C03656=1197.588,180.160,-56.490,-177.893,6.359,148.532
C03657=1197.583,180.408,-56.512,-177.890,6.361,148.532
C03658=1197.578,180.657,-56.536,-177.888,6.363,148.532
C03659=1197.574,180.906,-56.558,-177.885,6.365,148.531
C03660=1197.569,181.155,-56.581,-177.882,6.367,148.531
C03661=1197.565,181.403,-56.603,-177.880,6.368,148.531
C03662=1197.560,181.653,-56.626,-177.877,6.370,148.530
C03663=1197.555,181.902,-56.649,-177.874,6.372,148.530
C03664=1197.551,182.151,-56.672,-177.871,6.373,148.529
C03665=1197.546,182.400,-56.694,-177.868,6.375,148.529
C03666=1197.542,182.648,-56.717,-177.866,6.377,148.529
C03667=1197.537,182.898,-56.740,-177.864,6.378,148.528
C03668=1197.533,183.146,-56.763,-177.861,6.380,148.528
C03669=1197.527,183.395,-56.786,-177.858,6.382,148.527
C03670=1197.523,183.644,-56.809,-177.856,6.383,148.527
C03671=1197.519,183.893,-56.832,-177.853,6.385,148.527
C03672=1197.514,184.142,-56.855,-177.850,6.387,148.526
C03673=1197.509,184.392,-56.878,-177.848,6.389,148.526
C03674=1197.504,184.661,-56.902,-177.845,6.391,148.526
C03675=1197.499,184.930,-56.928,-177.842,6.393,148.525
C03676=1197.495,185.200,-56.952,-177.839,6.395,148.525
C03677=1197.489,185.469,-56.977,-177.836,6.397,148.525
C03678=1197.484,185.718,-57.000,-177.834,6.399,148.524
C03679=1197.480,185.967,-57.022,-177.831,6.400,148.524
C03680=1197.475,186.216,-57.046,-177.828,6.402,148.524
C03681=1197.470,186.465,-57.069,-177.826,6.404,148.523
C03682=1197.466,186.714,-57.092,-177.823,6.406,148.523
C03683=1197.462,186.963,-57.115,-177.820,6.408,148.523
C03684=1197.457,187.211,-57.138,-177.818,6.409,148.522
C03685=1197.452,187.460,-57.162,-177.815,6.411,148.522
C03686=1197.448,187.709,-57.184,-177.812,6.413,148.522
C03687=1197.443,187.958,-57.208,-177.810,6.415,148.521
C03688=1197.438,188.207,-57.231,-177.807,6.417,148.521
C03689=1197.434,188.456,-57.254,-177.805,6.419,148.520
C03690=1197.429,188.705,-57.278,-177.802,6.420,148.520
C03691=1197.424,188.953,-57.300,-177.799,6.422,148.520
C03692=1197.420,189.202,-57.324,-177.797,6.423,148.519
C03693=1197.415,189.451,-57.347,-177.794,6.425,148.519
C03694=1197.410,189.700,-57.370,-177.792,6.427,148.519
C03695=1197.406,189.949,-57.394,-177.789,6.429,148.518
C03696=1197.402,190.198,-57.416,-177.786,6.430,148.518
C03697=1197.397,190.447,-57.440,-177.784,6.432,148.518
C03698=1197.392,190.696,-57.463,-177.781,6.434,148.517
C03699=1197.388,190.945,-57.486,-177.779,6.436,148.517
C03700=1197.382,191.193,-57.509,-177.776,6.438,148.517
C03701=1197.378,191.442,-57.533,-177.774,6.440,148.516
C03702=1197.374,191.691,-57.556,-177.771,6.442,148.516
C03703=1197.369,191.940,-57.579,-177.768,6.443,148.516
C03704=1197.365,192.189,-57.603,-177.766,6.445,148.515
C03705=1197.360,192.438,-57.626,-177.763,6.447,148.515
C03706=1197.355,192.687,-57.650,-177.760,6.449,148.515
C03707=1197.350,192.936,-57.673,-177.758,6.451,148.514
C03708=1197.346,193.185,-57.696,-177.755,6.452,148.514
C03709=1197.341,193.434,-57.720,-177.752,6.454,148.514
C03710=1197.337,193.682,-57.744,-177.750,6.456,148.513
C03711=1197.332,193.931,-57.767,-177.747,6.458,148.513
C03712=1197.328,194.180,-57.790,-177.744,6.460,148.513
C03713=1197.323,194.429,-57.813,-177.742,6.461,148.512
C03714=1197.319,194.678,-57.837,-177.739,6.464,148.512
C03715=1197.314,194.926,-57.861,-177.736,6.466,148.512
C03716=1197.310,195.175,-57.884,-177.734,6.468,148.511
C03717=1197.305,195.425,-57.907,-177.731,6.470,148.511
C03718=1197.300,195.673,-57.932,-177.728,6.472,148.511
C03719=1197.296,195.922,-57.955,-177.726,6.473,148.510
C03720=1197.291,196.171,-57.978,-177.723,6.475,148.510
C03721=1197.287,196.419,-58.002,-177.720,6.477,148.510
C03722=1197.282,196.668,-58.026,-177.718,6.479,148.509
C03723=1197.277,196.917,-58.049,-177.715,6.481,148.509
C03724=1197.273,197.166,-58.073,-177.712,6.483,148.509
C03725=1197.268,197.415,-58.096,-177.710,6.484,148.508
C03726=1197.263,197.664,-58.120,-177.708,6.486,148.508
C03727=1197.259,197.912,-58.144,-177.705,6.488,148.508
C03728=1197.254,198.161,-58.167,-177.702,6.490,148.507
C03729=1197.250,198.410,-58.191,-177.700,6.492,148.507
C03730=1197.245,198.659,-58.215,-177.697,6.494,148.507
C03731=1197.240,198.908,-58.239,-177.694,6.496,148.506
C03732=1197.235,199.157,-58.263,-177.692,6.497,148.506
C03733=1197.231,199.406,-58.286,-177.689,6.499,148.506
C03734=1197.226,199.654,-58.310,-177.686,6.501,148.505
C03735=1197.222,199.904,-58.334,-177.684,6.503,148.505
C03736=1197.218,200.152,-58.358,-177.682,6.505,148.505
C03737=1197.213,200.401,-58.381,-177.679,6.507,148.505
C03738=1197.209,200.650,-58.405,-177.676,6.509,148.504
C03739=1197.204,200.899,-58.429,-177.673,6.511,148.504
C03740=1197.199,201.147,-58.453,-177.670,6.513,148.504
C03741=1197.194,201.396,-58.477,-177.668,6.515,148.503
C03742=1197.190,201.645,-58.501,-177.665,6.517,148.503
C03743=1197.185,201.893,-58.525,-177.662,6.518,148.503
C03744=1197.181,202.142,-58.548,-177.660,6.521,148.502
C03745=1197.177,202.391,-58.573,-177.658,6.522,148.502
C03746=1197.171,202.641,-58.597,-177.655,6.524,148.502
C03747=1197.167,202.889,-58.621,-177.652,6.526,148.501
C03748=1197.163,203.138,-58.645,-177.650,6.528,148.501
C03749=1197.158,203.387,-58.668,-177.647,6.530,148.501
C03750=1197.154,203.635,-58.692,-177.644,6.531,148.500
C03751=1197.149,203.884,-58.717,-177.642,6.534,148.500
C03752=1197.144,204.133,-58.741,-177.639,6.535,148.500
C03753=1197.140,204.382,-58.765,-177.636,6.538,148.500
C03754=1197.136,204.630,-58.789,-177.634,6.540,148.499
C03755=1197.130,204.880,-58.813,-177.631,6.542,148.499
C03756=1197.126,205.128,-58.837,-177.628,6.544,148.499
C03757=1197.122,205.377,-58.861,-177.626,6.545,148.498
C03758=1197.117,205.626,-58.885,-177.623,6.548,148.498
C03759=1197.112,205.875,-58.909,-177.621,6.549,148.498
C03760=1197.108,206.123,-58.933,-177.618,6.551,148.497
C03761=1197.103,206.372,-58.957,-177.615,6.553,148.497
C03762=1197.099,206.621,-58.983,-177.613,6.555,148.497
C03763=1197.094,206.870,-59.006,-177.610,6.557,148.496
C03764=1197.090,207.119,-59.030,-177.607,6.559,148.496
C03765=1197.085,207.367,-59.055,-177.605,6.561,148.496
C03766=1197.080,207.616,-59.079,-177.602,6.563,148.496
C03767=1197.076,207.865,-59.103,-177.599,6.565,148.495
C03768=1197.071,208.114,-59.127,-177.597,6.567,148.495
C03769=1197.067,208.363,-59.151,-177.594,6.569,148.495
C03770=1197.062,208.611,-59.175,-177.592,6.570,148.494
C03771=1197.058,208.860,-59.200,-177.589,6.573,148.494
C03772=1197.053,209.109,-59.224,-177.587,6.574,148.494
C03773=1197.048,209.358,-59.249,-177.583,6.577,148.494
C03774=1197.044,209.606,-59.273,-177.581,6.579,148.493
C03775=1197.040,209.855,-59.298,-177.578,6.581,148.493
C03776=1197.035,210.104,-59.322,-177.576,6.583,148.493
C03777=1197.030,210.352,-59.346,-177.573,6.585,148.492
C03778=1197.025,210.623,-59.372,-177.571,6.587,148.492
C03779=1197.020,210.894,-59.399,-177.568,6.589,148.492
C03780=1197.015,211.164,-59.426,-177.565,6.591,148.491
C03781=1197.010,211.434,-59.453,-177.562,6.594,148.491
C03782=1197.006,211.683,-59.477,-177.559,6.595,148.491
C03783=1197.002,211.932,-59.501,-177.556,6.597,148.490
C03784=1196.997,212.181,-59.526,-177.554,6.599,148.490
C03785=1196.992,212.429,-59.550,-177.552,6.601,148.490
C03786=1196.988,212.678,-59.575,-177.549,6.603,148.490
C03787=1196.983,212.927,-59.599,-177.546,6.606,148.489
C03788=1196.978,213.175,-59.624,-177.543,6.608,148.489
C03789=1196.975,213.425,-59.648,-177.540,6.609,148.489
C03790=1196.969,213.673,-59.673,-177.538,6.612,148.489
C03791=1196.965,213.921,-59.698,-177.536,6.613,148.488
C03792=1196.961,214.171,-59.723,-177.533,6.615,148.488
C03793=1196.956,214.419,-59.747,-177.530,6.617,148.488
C03794=1196.951,214.668,-59.771,-177.528,6.620,148.487
C03795=1196.947,214.917,-59.797,-177.525,6.622,148.487
C03796=1196.942,215.166,-59.821,-177.522,6.624,148.487
C03797=1196.938,215.415,-59.846,-177.520,6.625,148.486
C03798=1196.934,215.663,-59.870,-177.517,6.627,148.486
C03799=1196.929,215.911,-59.895,-177.515,6.629,148.486
C03800=1196.924,216.161,-59.920,-177.512,6.632,148.486
C03801=1196.920,216.409,-59.944,-177.509,6.634,148.485
C03802=1196.915,216.658,-59.970,-177.506,6.636,148.485
C03803=1196.911,216.907,-59.994,-177.504,6.638,148.485
C03804=1196.906,217.155,-60.019,-177.501,6.640,148.485
C03805=1196.901,217.405,-60.044,-177.499,6.642,148.484
C03806=1196.897,217.652,-60.069,-177.496,6.644,148.484
C03807=1196.893,217.902,-60.094,-177.493,6.646,148.484
C03808=1196.888,218.151,-60.118,-177.491,6.648,148.484
C03809=1196.884,218.398,-60.143,-177.488,6.650,148.483
C03810=1196.879,218.648,-60.168,-177.485,6.652,148.483
C03811=1196.874,218.897,-60.193,-177.483,6.654,148.483
C03812=1196.870,219.145,-60.218,-177.480,6.657,148.482
C03813=1196.865,219.394,-60.243,-177.477,6.658,148.482
C03814=1196.861,219.643,-60.268,-177.475,6.660,148.482
C03815=1196.857,219.891,-60.292,-177.473,6.662,148.482
C03816=1196.852,220.140,-60.317,-177.470,6.664,148.481
C03817=1196.847,220.388,-60.343,-177.467,6.667,148.481
C03818=1196.843,220.638,-60.368,-177.464,6.669,148.481
C03819=1196.839,220.886,-60.393,-177.462,6.671,148.481
C03820=1196.834,221.135,-60.418,-177.459,6.673,148.480
C03821=1196.829,221.384,-60.442,-177.457,6.675,148.480
C03822=1196.825,221.633,-60.468,-177.454,6.676,148.480
C03823=1196.820,221.881,-60.492,-177.451,6.679,148.480
C03824=1196.816,222.130,-60.518,-177.449,6.681,148.479
C03825=1196.811,222.379,-60.543,-177.446,6.683,148.479
C03826=1196.807,222.627,-60.568,-177.444,6.685,148.479
C03827=1196.802,222.876,-60.593,-177.441,6.687,148.478
C03828=1196.798,223.125,-60.618,-177.438,6.690,148.478
C03829=1196.793,223.373,-60.644,-177.435,6.691,148.478
C03830=1196.789,223.622,-60.669,-177.433,6.694,148.478
C03831=1196.784,223.870,-60.694,-177.431,6.695,148.477
C03832=1196.779,224.120,-60.719,-177.428,6.697,148.477
C03833=1196.775,224.368,-60.744,-177.425,6.700,148.477
C03834=1196.771,224.616,-60.770,-177.423,6.702,148.477
C03835=1196.766,224.865,-60.794,-177.420,6.704,148.476
C03836=1196.762,225.114,-60.820,-177.418,6.706,148.476
C03837=1196.757,225.363,-60.845,-177.415,6.708,148.476
C03838=1196.752,225.611,-60.870,-177.412,6.711,148.476
C03839=1196.748,225.860,-60.896,-177.409,6.712,148.475
C03840=1196.743,226.109,-60.921,-177.407,6.715,148.475
C03841=1196.739,226.358,-60.947,-177.404,6.716,148.475
C03842=1196.734,226.606,-60.972,-177.401,6.719,148.475
C03843=1196.731,226.854,-60.997,-177.399,6.721,148.474
C03844=1196.726,227.104,-61.022,-177.396,6.723,148.474
C03845=1196.721,227.352,-61.047,-177.394,6.725,148.474
C03846=1196.717,227.601,-61.073,-177.392,6.727,148.474
C03847=1196.712,227.849,-61.099,-177.388,6.730,148.473
C03848=1196.708,228.098,-61.124,-177.386,6.731,148.473
C03849=1196.703,228.347,-61.149,-177.384,6.734,148.473
C03850=1196.699,228.595,-61.175,-177.381,6.735,148.473
C03851=1196.694,228.844,-61.201,-177.378,6.738,148.472
C03852=1196.690,229.092,-61.226,-177.376,6.740,148.472
C03853=1196.685,229.341,-61.251,-177.373,6.742,148.472
C03854=1196.681,229.590,-61.277,-177.370,6.744,148.472
C03855=1196.676,229.838,-61.302,-177.368,6.747,148.471
C03856=1196.672,230.087,-61.328,-177.365,6.749,148.471
C03857=1196.667,230.336,-61.354,-177.362,6.751,148.471
C03858=1196.663,230.584,-61.379,-177.360,6.753,148.471
C03859=1196.658,230.833,-61.405,-177.358,6.755,148.470
C03860=1196.654,231.082,-61.430,-177.355,6.758,148.470
C03861=1196.649,231.330,-61.455,-177.352,6.759,148.470
C03862=1196.644,231.579,-61.482,-177.350,6.761,148.470
C03863=1196.640,231.828,-61.507,-177.347,6.763,148.470
C03864=1196.635,232.076,-61.533,-177.344,6.766,148.469
C03865=1196.631,232.325,-61.558,-177.342,6.768,148.469
C03866=1196.627,232.574,-61.584,-177.339,6.770,148.469
C03867=1196.622,232.823,-61.610,-177.337,6.772,148.469
C03868=1196.618,233.071,-61.635,-177.334,6.775,148.468
C03869=1196.613,233.320,-61.661,-177.331,6.777,148.468
C03870=1196.609,233.568,-61.687,-177.329,6.779,148.468
C03871=1196.604,233.817,-61.713,-177.327,6.781,148.468
C03872=1196.599,234.066,-61.739,-177.323,6.783,148.467
C03873=1196.595,234.315,-61.764,-177.321,6.785,148.467
C03874=1196.591,234.563,-61.791,-177.319,6.787,148.467
C03875=1196.586,234.811,-61.816,-177.315,6.790,148.467
C03876=1196.582,235.060,-61.842,-177.313,6.792,148.467
C03877=1196.577,235.309,-61.868,-177.311,6.794,148.466
C03878=1196.573,235.558,-61.894,-177.308,6.796,148.466
C03879=1196.568,235.806,-61.919,-177.305,6.799,148.466
C03880=1196.564,236.054,-61.945,-177.303,6.801,148.466
C03881=1196.560,236.303,-61.971,-177.300,6.803,148.465
C03882=1196.555,236.575,-62.000,-177.297,6.805,148.465
C03883=1196.549,236.846,-62.028,-177.295,6.807,148.465
C03884=1196.545,237.117,-62.057,-177.292,6.810,148.465
C03885=1196.540,237.389,-62.085,-177.289,6.813,148.465
C03886=1196.536,237.638,-62.110,-177.286,6.815,148.464
C03887=1196.531,237.886,-62.137,-177.284,6.817,148.464
C03888=1196.526,238.135,-62.163,-177.281,6.819,148.464
C03889=1196.522,238.383,-62.189,-177.278,6.821,148.464
C03890=1196.517,238.633,-62.215,-177.276,6.824,148.463
C03891=1196.513,238.881,-62.241,-177.273,6.825,148.463
C03892=1196.509,239.129,-62.267,-177.270,6.828,148.463
C03893=1196.504,239.378,-62.293,-177.268,6.830,148.463
C03894=1196.499,239.627,-62.319,-177.266,6.832,148.463
C03895=1196.495,239.875,-62.345,-177.263,6.834,148.462
C03896=1196.491,240.124,-62.371,-177.260,6.837,148.462
C03897=1196.486,240.373,-62.397,-177.258,6.839,148.462
C03898=1196.482,240.620,-62.424,-177.255,6.841,148.462
C03899=1196.477,240.869,-62.450,-177.252,6.844,148.462
C03900=1196.473,241.118,-62.476,-177.250,6.846,148.461
C03901=1196.469,241.366,-62.502,-177.248,6.848,148.461
C03902=1196.464,241.616,-62.528,-177.244,6.851,148.461
C03903=1196.460,241.864,-62.555,-177.242,6.853,148.461
C03904=1196.456,242.113,-62.581,-177.240,6.855,148.460
C03905=1196.451,242.361,-62.608,-177.237,6.858,148.460
C03906=1196.446,242.609,-62.633,-177.234,6.859,148.460
C03907=1196.441,242.858,-62.660,-177.232,6.862,148.460
C03908=1196.437,243.106,-62.686,-177.229,6.864,148.460
C03909=1196.432,243.355,-62.713,-177.227,6.866,148.460
C03910=1196.428,243.604,-62.739,-177.224,6.868,148.459
C03911=1196.424,243.852,-62.765,-177.222,6.870,148.459
C03912=1196.419,244.101,-62.792,-177.219,6.873,148.459
C03913=1196.415,244.349,-62.818,-177.217,6.875,148.459
C03914=1196.410,244.598,-62.844,-177.214,6.877,148.458
C03915=1196.407,244.847,-62.871,-177.211,6.880,148.458
C03916=1196.402,245.096,-62.897,-177.209,6.882,148.458
C03917=1196.398,245.344,-62.924,-177.206,6.884,148.458
C03918=1196.393,245.592,-62.951,-177.203,6.887,148.458
C03919=1196.388,245.840,-62.976,-177.201,6.889,148.457
C03920=1196.384,246.089,-63.003,-177.198,6.892,148.457
C03921=1196.379,246.338,-63.029,-177.195,6.893,148.457
C03922=1196.375,246.586,-63.056,-177.193,6.896,148.457
C03923=1196.370,246.835,-63.083,-177.190,6.898,148.457
C03924=1196.366,247.084,-63.109,-177.188,6.900,148.457
C03925=1196.361,247.332,-63.136,-177.186,6.903,148.456
C03926=1196.357,247.580,-63.162,-177.182,6.905,148.456
C03927=1196.352,247.829,-63.189,-177.180,6.907,148.456
C03928=1196.348,248.077,-63.215,-177.178,6.909,148.456
C03929=1196.344,248.326,-63.242,-177.175,6.912,148.456
C03930=1196.339,248.574,-63.269,-177.172,6.914,148.455
C03931=1196.335,248.823,-63.295,-177.170,6.916,148.455
C03932=1196.330,249.072,-63.322,-177.167,6.919,148.455
C03933=1196.326,249.320,-63.349,-177.165,6.921,148.455
C03934=1196.322,249.568,-63.376,-177.162,6.923,148.455
C03935=1196.317,249.817,-63.403,-177.159,6.926,148.455
C03936=1196.313,250.066,-63.428,-177.157,6.928,148.454
C03937=1196.308,250.314,-63.455,-177.154,6.931,148.454
C03938=1196.304,250.563,-63.483,-177.151,6.933,148.454
C03939=1196.300,250.812,-63.509,-177.149,6.935,148.454
C03940=1196.295,251.060,-63.536,-177.146,6.937,148.454
C03941=1196.291,251.309,-63.563,-177.144,6.940,148.453
C03942=1196.287,251.557,-63.589,-177.142,6.942,148.453
C03943=1196.282,251.806,-63.616,-177.138,6.944,148.453
C03944=1196.277,252.054,-63.643,-177.136,6.947,148.453
C03945=1196.273,252.303,-63.670,-177.133,6.949,148.453
C03946=1196.269,252.551,-63.697,-177.131,6.951,148.453
C03947=1196.264,252.800,-63.724,-177.128,6.953,148.452
C03948=1196.259,253.048,-63.751,-177.126,6.956,148.452
C03949=1196.255,253.297,-63.778,-177.123,6.958,148.452
C03950=1196.251,253.545,-63.805,-177.120,6.961,148.452
C03951=1196.247,253.794,-63.832,-177.118,6.963,148.452
C03952=1196.242,254.042,-63.859,-177.116,6.965,148.451
C03953=1196.237,254.291,-63.886,-177.113,6.968,148.451
C03954=1196.233,254.539,-63.913,-177.110,6.970,148.451
C03955=1196.229,254.788,-63.940,-177.107,6.973,148.451
C03956=1196.224,255.036,-63.967,-177.105,6.975,148.451
C03957=1196.219,255.285,-63.994,-177.103,6.977,148.451
C03958=1196.215,255.533,-64.021,-177.100,6.980,148.451
C03959=1196.212,255.782,-64.048,-177.097,6.982,148.450
C03960=1196.207,256.031,-64.075,-177.095,6.985,148.450
C03961=1196.202,256.278,-64.102,-177.092,6.987,148.450
C03962=1196.198,256.527,-64.130,-177.090,6.989,148.450
C03963=1196.193,256.775,-64.157,-177.087,6.992,148.450
C03964=1196.189,257.024,-64.184,-177.084,6.994,148.450
C03965=1196.184,257.273,-64.211,-177.082,6.997,148.449
C03966=1196.180,257.522,-64.238,-177.080,6.999,148.449
C03967=1196.176,257.770,-64.265,-177.076,7.002,148.449
C03968=1196.172,258.018,-64.292,-177.074,7.004,148.449
C03969=1196.167,258.266,-64.319,-177.072,7.006,148.449
C03970=1196.162,258.515,-64.347,-177.069,7.009,148.449
C03971=1196.158,258.764,-64.374,-177.067,7.011,148.449
C03972=1196.154,259.012,-64.402,-177.064,7.013,148.448
C03973=1196.149,259.260,-64.429,-177.061,7.016,148.448
C03974=1196.145,259.509,-64.456,-177.059,7.019,148.448
C03975=1196.140,259.758,-64.483,-177.056,7.020,148.448
C03976=1196.136,260.006,-64.511,-177.053,7.023,148.448
C03977=1196.131,260.254,-64.538,-177.051,7.025,148.448
C03978=1196.127,260.503,-64.565,-177.049,7.027,148.447
C03979=1196.122,260.751,-64.593,-177.046,7.030,148.447
C03980=1196.118,261.000,-64.620,-177.043,7.032,148.447
C03981=1196.114,261.248,-64.647,-177.041,7.035,148.447
C03982=1196.109,261.496,-64.675,-177.038,7.037,148.447
C03983=1196.105,261.745,-64.703,-177.035,7.040,148.447
C03984=1196.101,261.994,-64.730,-177.033,7.042,148.447
C03985=1196.096,262.242,-64.757,-177.030,7.045,148.447
C03986=1196.091,262.514,-64.788,-177.028,7.047,148.446
C03987=1196.087,262.787,-64.818,-177.025,7.050,148.446
C03988=1196.082,263.060,-64.848,-177.022,7.053,148.446
C03989=1196.077,263.333,-64.879,-177.019,7.056,148.446
C03990=1196.073,263.582,-64.906,-177.016,7.058,148.446
C03991=1196.068,263.830,-64.933,-177.014,7.061,148.446
C03992=1196.064,264.078,-64.961,-177.012,7.063,148.445
C03993=1196.059,264.327,-64.988,-177.008,7.066,148.445
C03994=1196.055,264.575,-65.016,-177.006,7.068,148.445
C03995=1196.051,264.823,-65.044,-177.004,7.071,148.445
C03996=1196.047,265.072,-65.071,-177.001,7.073,148.445
C03997=1196.042,265.320,-65.099,-176.998,7.076,148.445
C03998=1196.037,265.569,-65.127,-176.996,7.078,148.445
C03999=1196.033,265.818,-65.155,-176.993,7.080,148.444
C04000=1196.029,266.066,-65.182,-176.991,7.083,148.444
C04001=1196.024,266.314,-65.210,-176.989,7.085,148.444
C04002=1196.020,266.563,-65.238,-176.986,7.088,148.444
C04003=1196.016,266.811,-65.265,-176.983,7.090,148.444
C04004=1196.011,267.059,-65.293,-176.981,7.093,148.444
C04005=1196.007,267.308,-65.321,-176.978,7.095,148.444
C04006=1196.002,267.556,-65.348,-176.975,7.097,148.443
C04007=1195.999,267.805,-65.377,-176.973,7.100,148.443
C04008=1195.993,268.054,-65.404,-176.970,7.103,148.443
C04009=1195.989,268.302,-65.432,-176.968,7.104,148.443
C04010=1195.985,268.550,-65.460,-176.965,7.107,148.443
C04011=1195.981,268.798,-65.488,-176.963,7.110,148.443
C04012=1195.977,269.047,-65.515,-176.960,7.113,148.443
C04013=1195.972,269.295,-65.544,-176.958,7.115,148.443
C04014=1195.967,269.543,-65.571,-176.955,7.118,148.443
C04015=1195.963,269.792,-65.600,-176.953,7.120,148.442
C04016=1195.958,270.041,-65.627,-176.950,7.123,148.442
C04017=1195.954,270.289,-65.655,-176.947,7.125,148.442
C04018=1195.950,270.537,-65.683,-176.945,7.128,148.442
C04019=1195.945,270.785,-65.712,-176.942,7.131,148.442
C04020=1195.941,271.034,-65.740,-176.939,7.132,148.442
C04021=1195.936,271.282,-65.767,-176.937,7.135,148.442
C04022=1195.933,271.531,-65.795,-176.934,7.138,148.442
C04023=1195.928,271.779,-65.823,-176.932,7.141,148.442
C04024=1195.924,272.028,-65.851,-176.929,7.142,148.441
C04025=1195.919,272.276,-65.880,-176.926,7.145,148.441
C04026=1195.915,272.524,-65.908,-176.924,7.148,148.441
C04027=1195.911,272.772,-65.936,-176.922,7.151,148.441
C04028=1195.906,273.021,-65.964,-176.919,7.152,148.441
C04029=1195.902,273.269,-65.992,-176.916,7.155,148.441
C04030=1195.898,273.518,-66.020,-176.914,7.158,148.441
C04031=1195.893,273.766,-66.049,-176.911,7.161,148.441
C04032=1195.889,274.014,-66.077,-176.909,7.163,148.440
C04033=1195.884,274.263,-66.105,-176.906,7.166,148.440
C04034=1195.880,274.511,-66.133,-176.904,7.168,148.440
C04035=1195.875,274.759,-66.162,-176.901,7.171,148.440
C04036=1195.872,275.008,-66.190,-176.898,7.174,148.440
C04037=1195.867,275.256,-66.218,-176.896,7.176,148.440
C04038=1195.863,275.505,-66.246,-176.893,7.179,148.440
C04039=1195.858,275.753,-66.274,-176.891,7.181,148.440
C04040=1195.854,276.002,-66.303,-176.888,7.184,148.440
C04041=1195.850,276.249,-66.331,-176.886,7.186,148.439
C04042=1195.845,276.498,-66.359,-176.883,7.189,148.439
C04043=1195.841,276.746,-66.387,-176.881,7.191,148.439
C04044=1195.836,276.995,-66.416,-176.878,7.194,148.439
C04045=1195.833,277.244,-66.444,-176.875,7.197,148.439
C04046=1195.828,277.491,-66.473,-176.873,7.199,148.439
C04047=1195.824,277.740,-66.501,-176.870,7.202,148.439
C04048=1195.819,277.988,-66.530,-176.868,7.204,148.439
C04049=1195.815,278.237,-66.558,-176.865,7.207,148.439
C04050=1195.810,278.485,-66.586,-176.863,7.209,148.439
C04051=1195.806,278.734,-66.615,-176.860,7.212,148.439
C04052=1195.802,278.982,-66.644,-176.857,7.215,148.438
C04053=1195.797,279.230,-66.672,-176.855,7.217,148.438
C04054=1195.793,279.478,-66.700,-176.852,7.220,148.438
C04055=1195.789,279.727,-66.729,-176.850,7.222,148.438
C04056=1195.784,279.975,-66.758,-176.847,7.225,148.438
C04057=1195.780,280.223,-66.786,-176.845,7.227,148.438
C04058=1195.775,280.472,-66.815,-176.842,7.230,148.438
C04059=1195.772,280.719,-66.844,-176.839,7.233,148.438
C04060=1195.767,280.968,-66.872,-176.837,7.235,148.438
C04061=1195.762,281.217,-66.901,-176.835,7.238,148.438
C04062=1195.759,281.465,-66.929,-176.832,7.240,148.438
C04063=1195.754,281.713,-66.958,-176.829,7.243,148.437
C04064=1195.749,281.962,-66.987,-176.827,7.245,148.437
C04065=1195.746,282.210,-67.015,-176.824,7.248,148.437
C04066=1195.741,282.458,-67.044,-176.822,7.251,148.437
C04067=1195.736,282.706,-67.073,-176.820,7.253,148.437
C04068=1195.733,282.955,-67.101,-176.817,7.256,148.437
C04069=1195.728,283.203,-67.130,-176.815,7.259,148.437
C04070=1195.723,283.451,-67.159,-176.811,7.261,148.437
C04071=1195.719,283.700,-67.188,-176.809,7.264,148.437
C04072=1195.715,283.948,-67.217,-176.807,7.266,148.437
C04073=1195.710,284.196,-67.245,-176.804,7.269,148.437
C04074=1195.706,284.444,-67.275,-176.802,7.272,148.437
C04075=1195.702,284.693,-67.303,-176.799,7.275,148.437
C04076=1195.698,284.940,-67.332,-176.796,7.278,148.437
C04077=1195.693,285.189,-67.361,-176.794,7.280,148.437
C04078=1195.689,285.438,-67.390,-176.791,7.282,148.436
C04079=1195.685,285.687,-67.419,-176.788,7.285,148.436
C04080=1195.680,285.934,-67.448,-176.786,7.288,148.436
C04081=1195.676,286.182,-67.477,-176.783,7.291,148.436
C04082=1195.672,286.431,-67.506,-176.781,7.293,148.436
C04083=1195.668,286.679,-67.535,-176.779,7.296,148.436
C04084=1195.663,286.927,-67.563,-176.776,7.299,148.436
C04085=1195.658,287.176,-67.593,-176.774,7.301,148.436
C04086=1195.654,287.424,-67.622,-176.771,7.304,148.436
C04087=1195.650,287.672,-67.650,-176.769,7.306,148.436
C04088=1195.646,287.920,-67.679,-176.766,7.309,148.436
C04089=1195.641,288.168,-67.709,-176.763,7.312,148.436
C04090=1195.637,288.443,-67.741,-176.760,7.315,148.436
C04091=1195.632,288.718,-67.773,-176.758,7.318,148.436
C04092=1195.627,288.992,-67.806,-176.755,7.321,148.436
C04093=1195.622,289.266,-67.837,-176.752,7.324,148.435
C04094=1195.618,289.514,-67.867,-176.750,7.326,148.435
C04095=1195.614,289.763,-67.896,-176.747,7.329,148.435
C04096=1195.610,290.012,-67.925,-176.744,7.332,148.435
C04097=1195.605,290.260,-67.954,-176.742,7.334,148.435
C04098=1195.601,290.507,-67.983,-176.739,7.337,148.435
C04099=1195.596,290.756,-68.013,-176.737,7.340,148.435
C04100=1195.592,291.004,-68.042,-176.735,7.342,148.435
C04101=1195.588,291.253,-68.071,-176.732,7.345,148.435
C04102=1195.584,291.501,-68.100,-176.729,7.348,148.435
C04103=1195.579,291.749,-68.130,-176.727,7.350,148.435
C04104=1195.575,291.997,-68.159,-176.724,7.353,148.435
C04105=1195.570,292.245,-68.188,-176.722,7.356,148.435
C04106=1195.566,292.493,-68.218,-176.719,7.359,148.435
C04107=1195.562,292.742,-68.247,-176.717,7.362,148.435
C04108=1195.558,292.990,-68.277,-176.715,7.364,148.435
C04109=1195.554,293.238,-68.306,-176.712,7.367,148.435
C04110=1195.549,293.487,-68.336,-176.709,7.370,148.435
C04111=1195.545,293.735,-68.365,-176.707,7.372,148.435
C04112=1195.541,293.982,-68.394,-176.704,7.375,148.435
C04113=1195.536,294.231,-68.424,-176.702,7.378,148.434
C04114=1195.532,294.479,-68.453,-176.699,7.380,148.434
C04115=1195.528,294.727,-68.483,-176.697,7.383,148.434
C04116=1195.524,294.975,-68.512,-176.694,7.386,148.434
C04117=1195.519,295.224,-68.542,-176.692,7.388,148.434
C04118=1195.515,295.472,-68.572,-176.689,7.391,148.434
C04119=1195.511,295.721,-68.601,-176.686,7.394,148.434
C04120=1195.506,295.969,-68.630,-176.684,7.397,148.434
C04121=1195.502,296.217,-68.660,-176.682,7.400,148.434
C04122=1195.498,296.465,-68.689,-176.679,7.403,148.434
C04123=1195.494,296.714,-68.719,-176.677,7.405,148.434
C04124=1195.490,296.962,-68.748,-176.674,7.408,148.434
C04125=1195.485,297.210,-68.778,-176.671,7.411,148.434
C04126=1195.481,297.458,-68.809,-176.669,7.413,148.434
C04127=1195.477,297.706,-68.838,-176.667,7.416,148.434
C04128=1195.472,297.954,-68.867,-176.664,7.419,148.434
C04129=1195.468,298.202,-68.897,-176.661,7.422,148.434
C04130=1195.463,298.451,-68.927,-176.659,7.424,148.434
C04131=1195.459,298.698,-68.957,-176.656,7.427,148.434
C04132=1195.455,298.947,-68.986,-176.654,7.430,148.434
C04133=1195.451,299.195,-69.016,-176.651,7.432,148.434
C04134=1195.446,299.443,-69.045,-176.649,7.435,148.434
C04135=1195.442,299.691,-69.076,-176.646,7.438,148.434
C04136=1195.438,299.939,-69.105,-176.644,7.441,148.434
C04137=1195.433,300.188,-69.135,-176.641,7.444,148.434
C04138=1195.428,300.436,-69.165,-176.639,7.447,148.434
C04139=1195.425,300.684,-69.195,-176.636,7.449,148.434
C04140=1195.421,300.933,-69.225,-176.634,7.452,148.434
C04141=1195.417,301.181,-69.254,-176.631,7.455,148.434
C04142=1195.412,301.429,-69.285,-176.629,7.458,148.434
C04143=1195.408,301.677,-69.314,-176.627,7.460,148.434
C04144=1195.404,301.925,-69.345,-176.624,7.463,148.434
C04145=1195.399,302.174,-69.375,-176.621,7.466,148.434
C04146=1195.395,302.422,-69.404,-176.619,7.469,148.434
C04147=1195.391,302.670,-69.434,-176.616,7.472,148.434
C04148=1195.386,302.918,-69.464,-176.614,7.475,148.434
C04149=1195.382,303.166,-69.495,-176.612,7.477,148.433
C04150=1195.378,303.414,-69.524,-176.609,7.480,148.433
C04151=1195.374,303.662,-69.555,-176.606,7.483,148.433
C04152=1195.369,303.910,-69.584,-176.603,7.486,148.433
C04153=1195.364,304.159,-69.614,-176.602,7.488,148.434
C04154=1195.361,304.407,-69.644,-176.599,7.491,148.434
C04155=1195.356,304.655,-69.674,-176.596,7.494,148.434
C04156=1195.352,304.903,-69.705,-176.594,7.497,148.433
C04157=1195.349,305.151,-69.735,-176.591,7.500,148.433
C04158=1195.344,305.400,-69.765,-176.589,7.503,148.433
C04159=1195.340,305.647,-69.795,-176.586,7.506,148.433
C04160=1195.335,305.896,-69.825,-176.584,7.508,148.433
C04161=1195.331,306.144,-69.856,-176.582,7.511,148.434
C04162=1195.326,306.392,-69.886,-176.579,7.514,148.434
C04163=1195.322,306.640,-69.916,-176.577,7.516,148.433
C04164=1195.318,306.888,-69.947,-176.574,7.519,148.433
C04165=1195.314,307.137,-69.976,-176.571,7.522,148.433
C04166=1195.309,307.385,-70.007,-176.569,7.525,148.433
C04167=1195.305,307.632,-70.037,-176.567,7.528,148.434
C04168=1195.301,307.881,-70.067,-176.564,7.531,148.434
C04169=1195.297,308.129,-70.098,-176.562,7.534,148.434
C04170=1195.293,308.377,-70.129,-176.559,7.537,148.434
C04171=1195.288,308.625,-70.158,-176.557,7.539,148.433
C04172=1195.284,308.873,-70.189,-176.554,7.542,148.433
C04173=1195.280,309.121,-70.219,-176.552,7.545,148.434
C04174=1195.275,309.369,-70.250,-176.550,7.548,148.434
C04175=1195.270,309.618,-70.280,-176.547,7.551,148.434
C04176=1195.267,309.866,-70.310,-176.544,7.554,148.434
C04177=1195.263,310.114,-70.341,-176.542,7.557,148.434
C04178=1195.259,310.362,-70.371,-176.540,7.559,148.434
C04179=1195.254,310.609,-70.402,-176.537,7.562,148.434
C04180=1195.250,310.858,-70.433,-176.535,7.565,148.434
C04181=1195.246,311.106,-70.463,-176.532,7.568,148.434
C04182=1195.241,311.354,-70.493,-176.530,7.570,148.434
C04183=1195.237,311.602,-70.524,-176.528,7.574,148.434
C04184=1195.233,311.850,-70.554,-176.525,7.577,148.434
C04185=1195.229,312.099,-70.586,-176.522,7.580,148.434
C04186=1195.225,312.346,-70.616,-176.520,7.582,148.434
C04187=1195.220,312.594,-70.646,-176.518,7.585,148.434
C04188=1195.216,312.842,-70.677,-176.515,7.588,148.434
C04189=1195.212,313.091,-70.708,-176.512,7.591,148.434
C04190=1195.208,313.339,-70.739,-176.510,7.593,148.434
C04191=1195.203,313.586,-70.769,-176.508,7.597,148.434
C04192=1195.199,313.835,-70.800,-176.505,7.600,148.434
C04193=1195.195,314.083,-70.831,-176.503,7.602,148.434
C04194=1195.190,314.359,-70.864,-176.500,7.606,148.434
C04195=1195.185,314.636,-70.899,-176.497,7.609,148.434
C04196=1195.180,314.912,-70.933,-176.495,7.612,148.434
C04197=1195.176,315.189,-70.968,-176.492,7.615,148.434
C04198=1195.171,315.437,-70.998,-176.490,7.618,148.434
C04199=1195.168,315.685,-71.029,-176.487,7.621,148.434
C04200=1195.163,315.933,-71.060,-176.485,7.624,148.434
C04201=1195.159,316.181,-71.090,-176.482,7.627,148.434
C04202=1195.155,316.428,-71.122,-176.480,7.630,148.434
C04203=1195.151,316.677,-71.152,-176.478,7.633,148.435
C04204=1195.147,316.925,-71.183,-176.475,7.635,148.435
C04205=1195.142,317.173,-71.214,-176.473,7.638,148.435
C04206=1195.138,317.421,-71.245,-176.470,7.641,148.435
C04207=1195.133,317.669,-71.276,-176.468,7.645,148.435
C04208=1195.129,317.917,-71.307,-176.465,7.648,148.435
C04209=1195.126,318.165,-71.338,-176.463,7.650,148.435
C04210=1195.121,318.413,-71.369,-176.461,7.653,148.435
C04211=1195.117,318.662,-71.400,-176.458,7.656,148.435
C04212=1195.113,318.910,-71.431,-176.455,7.659,148.435
C04213=1195.108,319.157,-71.462,-176.454,7.662,148.435
C04214=1195.104,319.406,-71.493,-176.451,7.665,148.435
C04215=1195.100,319.654,-71.524,-176.449,7.668,148.435
C04216=1195.095,319.901,-71.555,-176.446,7.671,148.435
C04217=1195.092,320.149,-71.586,-176.444,7.673,148.435
C04218=1195.088,320.397,-71.617,-176.442,7.677,148.435
C04219=1195.084,320.645,-71.649,-176.439,7.680,148.435
C04220=1195.079,320.893,-71.679,-176.436,7.683,148.435
C04221=1195.075,321.142,-71.710,-176.435,7.685,148.436
C04222=1195.071,321.389,-71.742,-176.432,7.688,148.436
C04223=1195.066,321.637,-71.773,-176.430,7.691,148.436
C04224=1195.062,321.886,-71.804,-176.427,7.694,148.436
C04225=1195.058,322.133,-71.835,-176.424,7.698,148.436
C04226=1195.054,322.382,-71.866,-176.423,7.700,148.436
C04227=1195.050,322.629,-71.898,-176.420,7.703,148.436
C04228=1195.046,322.878,-71.929,-176.418,7.706,148.436
C04229=1195.041,323.125,-71.960,-176.415,7.709,148.436
C04230=1195.037,323.374,-71.992,-176.413,7.712,148.436
C04231=1195.033,323.621,-72.023,-176.411,7.715,148.436
C04232=1195.029,323.870,-72.054,-176.408,7.718,148.436
C04233=1195.025,324.117,-72.086,-176.406,7.721,148.436
C04234=1195.021,324.366,-72.117,-176.403,7.724,148.436
C04235=1195.016,324.613,-72.148,-176.401,7.727,148.437
C04236=1195.012,324.862,-72.179,-176.399,7.730,148.437
C04237=1195.008,325.109,-72.211,-176.396,7.733,148.437
C04238=1195.004,325.358,-72.242,-176.394,7.736,148.437
C04239=1195.000,325.605,-72.274,-176.392,7.739,148.437
C04240=1194.995,325.854,-72.305,-176.389,7.742,148.437
C04241=1194.991,326.101,-72.337,-176.387,7.745,148.437
C04242=1194.987,326.349,-72.369,-176.384,7.748,148.437
C04243=1194.982,326.597,-72.399,-176.382,7.751,148.437
C04244=1194.979,326.845,-72.431,-176.380,7.754,148.437
C04245=1194.974,327.093,-72.463,-176.378,7.757,148.438
C04246=1194.970,327.341,-72.494,-176.375,7.760,148.438
C04247=1194.967,327.590,-72.526,-176.373,7.763,148.438
C04248=1194.962,327.837,-72.558,-176.371,7.765,148.438
C04249=1194.958,328.086,-72.589,-176.368,7.769,148.438
C04250=1194.953,328.333,-72.620,-176.366,7.772,148.438
C04251=1194.950,328.581,-72.652,-176.364,7.775,148.438
C04252=1194.945,328.829,-72.684,-176.361,7.778,148.438
C04253=1194.940,329.078,-72.715,-176.359,7.781,148.438
C04254=1194.937,329.326,-72.747,-176.356,7.784,148.438
C04255=1194.932,329.573,-72.779,-176.354,7.787,148.439
C04256=1194.929,329.821,-72.811,-176.352,7.790,148.439
C04257=1194.924,330.069,-72.843,-176.349,7.793,148.439
C04258=1194.920,330.317,-72.874,-176.348,7.796,148.439
C04259=1194.915,330.565,-72.905,-176.345,7.799,148.439
C04260=1194.912,330.813,-72.937,-176.343,7.802,148.439
C04261=1194.907,331.061,-72.970,-176.340,7.805,148.439
C04262=1194.903,331.308,-73.001,-176.338,7.808,148.439
C04263=1194.899,331.556,-73.033,-176.336,7.811,148.440
C04264=1194.896,331.804,-73.065,-176.333,7.814,148.440
C04265=1194.890,332.053,-73.096,-176.331,7.817,148.440
C04266=1194.886,332.301,-73.128,-176.328,7.820,148.440
C04267=1194.883,332.549,-73.160,-176.327,7.823,148.440
C04268=1194.878,332.796,-73.192,-176.325,7.826,148.440
C04269=1194.874,333.044,-73.224,-176.322,7.829,148.440
C04270=1194.870,333.292,-73.255,-176.320,7.833,148.440
C04271=1194.865,333.540,-73.288,-176.317,7.836,148.441
C04272=1194.862,333.788,-73.319,-176.315,7.838,148.441
C04273=1194.858,334.036,-73.351,-176.313,7.841,148.441
C04274=1194.853,334.284,-73.383,-176.311,7.845,148.441
C04275=1194.849,334.532,-73.415,-176.308,7.848,148.441
C04276=1194.845,334.780,-73.448,-176.306,7.851,148.441
C04277=1194.840,335.028,-73.479,-176.304,7.854,148.441
C04278=1194.837,335.276,-73.511,-176.301,7.857,148.441
C04279=1194.832,335.523,-73.544,-176.299,7.860,148.442
C04280=1194.828,335.771,-73.576,-176.297,7.863,148.442
C04281=1194.824,336.019,-73.608,-176.295,7.867,148.442
C04282=1194.820,336.267,-73.640,-176.293,7.869,148.442
C04283=1194.816,336.515,-73.672,-176.290,7.872,148.442
C04284=1194.811,336.763,-73.704,-176.288,7.875,148.442
C04285=1194.808,337.011,-73.736,-176.285,7.878,148.442
C04286=1194.803,337.259,-73.769,-176.284,7.881,148.443
C04287=1194.799,337.506,-73.800,-176.282,7.884,148.443
C04288=1194.795,337.754,-73.833,-176.279,7.888,148.443
C04289=1194.791,338.002,-73.865,-176.277,7.891,148.443
C04290=1194.787,338.251,-73.897,-176.274,7.894,148.443
C04291=1194.783,338.497,-73.929,-176.273,7.896,148.443
C04292=1194.778,338.746,-73.962,-176.270,7.900,148.444
C04293=1194.774,338.994,-73.993,-176.268,7.903,148.444
C04294=1194.770,339.242,-74.026,-176.266,7.906,148.444
C04295=1194.767,339.489,-74.058,-176.263,7.909,148.444
C04296=1194.761,339.737,-74.091,-176.262,7.912,148.444
C04297=1194.758,339.985,-74.122,-176.259,7.915,148.444
C04298=1194.753,340.264,-74.159,-176.257,7.919,148.445
C04299=1194.749,340.542,-74.196,-176.254,7.923,148.445
C04300=1194.744,340.821,-74.233,-176.252,7.926,148.445
C04301=1194.738,341.100,-74.268,-176.249,7.929,148.445
C04302=1194.735,341.347,-74.301,-176.247,7.932,148.445
C04303=1194.730,341.595,-74.333,-176.245,7.936,148.446
C04304=1194.727,341.843,-74.366,-176.243,7.939,148.446
C04305=1194.723,342.091,-74.398,-176.241,7.942,148.446
C04306=1194.718,342.339,-74.430,-176.239,7.945,148.446
C04307=1194.714,342.586,-74.463,-176.237,7.948,148.446
C04308=1194.710,342.835,-74.495,-176.234,7.951,148.446
C04309=1194.706,343.082,-74.528,-176.232,7.955,148.447
C04310=1194.702,343.330,-74.560,-176.230,7.957,148.447
C04311=1194.698,343.578,-74.593,-176.228,7.960,148.447
C04312=1194.693,343.826,-74.625,-176.226,7.964,148.447
C04313=1194.689,344.073,-74.658,-176.223,7.967,148.448
C04314=1194.685,344.321,-74.690,-176.221,7.970,148.448
C04315=1194.681,344.569,-74.724,-176.219,7.973,148.448
C04316=1194.677,344.817,-74.755,-176.217,7.976,148.448
C04317=1194.673,345.065,-74.789,-176.215,7.980,148.448
C04318=1194.668,345.313,-74.821,-176.213,7.983,148.449
C04319=1194.664,345.561,-74.854,-176.210,7.986,148.449
C04320=1194.660,345.808,-74.886,-176.209,7.989,148.449
C04321=1194.656,346.056,-74.919,-176.207,7.992,148.449
C04322=1194.652,346.304,-74.952,-176.204,7.995,148.449
C04323=1194.647,346.552,-74.984,-176.202,7.999,148.450
C04324=1194.644,346.800,-75.017,-176.200,8.002,148.450
C04325=1194.640,347.047,-75.050,-176.198,8.005,148.450
C04326=1194.635,347.296,-75.083,-176.196,8.008,148.450
C04327=1194.631,347.543,-75.116,-176.194,8.011,148.450
C04328=1194.627,347.791,-75.149,-176.191,8.015,148.451
C04329=1194.624,348.039,-75.181,-176.189,8.018,148.451
C04330=1194.619,348.287,-75.214,-176.188,8.020,148.451
C04331=1194.615,348.535,-75.247,-176.185,8.024,148.451
C04332=1194.611,348.782,-75.280,-176.184,8.027,148.452
C04333=1194.606,349.029,-75.313,-176.181,8.031,148.452
C04334=1194.602,349.278,-75.345,-176.180,8.033,148.452
C04335=1194.598,349.525,-75.378,-176.177,8.037,148.452
C04336=1194.594,349.773,-75.411,-176.175,8.040,148.453
C04337=1194.590,350.021,-75.444,-176.173,8.043,148.453
C04338=1194.586,350.269,-75.477,-176.171,8.046,148.453
C04339=1194.581,350.517,-75.510,-176.169,8.049,148.453
C04340=1194.577,350.764,-75.543,-176.167,8.053,148.454
C04341=1194.573,351.012,-75.576,-176.165,8.056,148.454
C04342=1194.569,351.260,-75.609,-176.163,8.059,148.454
C04343=1194.565,351.508,-75.643,-176.160,8.063,148.454
C04344=1194.561,351.755,-75.676,-176.159,8.065,148.454
C04345=1194.557,352.003,-75.708,-176.157,8.069,148.455
C04346=1194.553,352.251,-75.741,-176.155,8.072,148.455
C04347=1194.549,352.499,-75.774,-176.153,8.075,148.455
C04348=1194.545,352.747,-75.807,-176.150,8.079,148.456
C04349=1194.540,352.994,-75.840,-176.149,8.082,148.456
C04350=1194.536,353.242,-75.873,-176.147,8.085,148.456
C04351=1194.532,353.490,-75.907,-176.145,8.088,148.456
C04352=1194.528,353.737,-75.940,-176.142,8.092,148.457
C04353=1194.525,353.986,-75.973,-176.141,8.094,148.457
C04354=1194.520,354.234,-76.006,-176.139,8.098,148.457
C04355=1194.516,354.481,-76.039,-176.137,8.101,148.457
C04356=1194.512,354.729,-76.073,-176.135,8.105,148.458
C04357=1194.508,354.977,-76.106,-176.133,8.108,148.458
C04358=1194.504,355.225,-76.139,-176.131,8.110,148.458
C04359=1194.500,355.472,-76.172,-176.129,8.114,148.459
C04360=1194.496,355.719,-76.206,-176.127,8.117,148.459
C04361=1194.492,355.967,-76.239,-176.125,8.121,148.459
C04362=1194.488,356.215,-76.272,-176.123,8.124,148.460
C04363=1194.483,356.463,-76.305,-176.121,8.127,148.460
C04364=1194.479,356.710,-76.339,-176.119,8.130,148.460
C04365=1194.474,356.958,-76.372,-176.117,8.134,148.460
C04366=1194.471,357.207,-76.406,-176.115,8.137,148.461
C04367=1194.467,357.455,-76.439,-176.114,8.140,148.461
C04368=1194.463,357.702,-76.473,-176.112,8.143,148.461
C04369=1194.459,357.949,-76.506,-176.110,8.147,148.462
C04370=1194.455,358.197,-76.539,-176.108,8.150,148.462
C04371=1194.451,358.445,-76.572,-176.106,8.154,148.462
C04372=1194.446,358.693,-76.606,-176.104,8.156,148.463
C04373=1194.443,358.940,-76.639,-176.102,8.160,148.463
C04374=1194.438,359.188,-76.674,-176.100,8.163,148.463
C04375=1194.434,359.436,-76.707,-176.098,8.167,148.464
C04376=1194.430,359.684,-76.740,-176.097,8.170,148.464
C04377=1194.426,359.931,-76.774,-176.095,8.173,148.464
C04378=1194.422,360.179,-76.807,-176.093,8.176,148.465
C04379=1194.418,360.426,-76.840,-176.091,8.179,148.465
C04380=1194.415,360.674,-76.874,-176.089,8.183,148.465
C04381=1194.410,360.922,-76.908,-176.087,8.186,148.466
C04382=1194.406,361.170,-76.941,-176.086,8.190,148.466
C04383=1194.402,361.417,-76.975,-176.084,8.192,148.466
C04384=1194.398,361.665,-77.008,-176.082,8.196,148.467
C04385=1194.393,361.913,-77.042,-176.080,8.199,148.467
C04386=1194.390,362.161,-77.076,-176.079,8.202,148.467
C04387=1194.385,362.408,-77.109,-176.077,8.206,148.468
C04388=1194.382,362.656,-77.143,-176.075,8.209,148.468
C04389=1194.377,362.903,-77.176,-176.073,8.213,148.468
C04390=1194.373,363.151,-77.211,-176.072,8.216,148.469
C04391=1194.369,363.399,-77.244,-176.070,8.219,148.469
C04392=1194.365,363.647,-77.278,-176.068,8.222,148.469
C04393=1194.361,363.894,-77.311,-176.066,8.225,148.470
C04394=1194.357,364.142,-77.345,-176.064,8.229,148.470
C04395=1194.353,364.390,-77.379,-176.063,8.232,148.471
C04396=1194.349,364.638,-77.413,-176.061,8.235,148.471
C04397=1194.345,364.885,-77.447,-176.059,8.239,148.471
C04398=1194.340,365.133,-77.480,-176.058,8.242,148.472
C04399=1194.337,365.380,-77.514,-176.056,8.245,148.472
C04400=1194.333,365.628,-77.549,-176.054,8.249,148.473
C04401=1194.328,365.876,-77.582,-176.053,8.252,148.473
C04402=1194.324,366.157,-77.621,-176.051,8.255,148.473
C04403=1194.320,366.438,-77.659,-176.050,8.259,148.474
C04404=1194.315,366.719,-77.697,-176.048,8.262,148.474
C04405=1194.310,366.999,-77.736,-176.045,8.267,148.475
C04406=1194.307,367.247,-77.770,-176.044,8.270,148.475
C04407=1194.303,367.494,-77.804,-176.042,8.273,148.476
C04408=1194.298,367.742,-77.837,-176.041,8.276,148.476
C04409=1194.295,367.990,-77.872,-176.039,8.280,148.476
C04410=1194.290,368.238,-77.905,-176.038,8.283,148.477
C04411=1194.286,368.485,-77.939,-176.036,8.286,148.477
C04412=1194.282,368.732,-77.973,-176.035,8.289,148.478
C04413=1194.278,368.981,-78.007,-176.033,8.293,148.478
C04414=1194.274,369.228,-78.041,-176.032,8.295,148.478
C04415=1194.269,369.476,-78.076,-176.030,8.299,148.479
C04416=1194.266,369.724,-78.110,-176.029,8.302,148.479
C04417=1194.261,369.972,-78.144,-176.027,8.306,148.480
C04418=1194.258,370.219,-78.178,-176.026,8.308,148.480
C04419=1194.254,370.467,-78.212,-176.024,8.312,148.480
C04420=1194.250,370.714,-78.246,-176.023,8.315,148.481
C04421=1194.245,370.962,-78.280,-176.021,8.318,148.481
C04422=1194.242,371.210,-78.314,-176.020,8.321,148.482
C04423=1194.238,371.457,-78.348,-176.019,8.325,148.482
C04424=1194.233,371.704,-78.383,-176.018,8.328,148.483
C04425=1194.230,371.952,-78.417,-176.016,8.332,148.483
C04426=1194.225,372.200,-78.451,-176.015,8.334,148.484
C04427=1194.221,372.447,-78.484,-176.013,8.337,148.484
C04428=1194.217,372.695,-78.519,-176.012,8.341,148.485
C04429=1194.213,372.943,-78.554,-176.011,8.344,148.485
C04430=1194.209,373.191,-78.588,-176.009,8.348,148.485
C04431=1194.205,373.438,-78.622,-176.008,8.350,148.486
C04432=1194.201,373.685,-78.656,-176.007,8.353,148.486
C04433=1194.197,373.933,-78.691,-176.005,8.357,148.487
C04434=1194.193,374.181,-78.724,-176.004,8.360,148.487
C04435=1194.188,374.428,-78.759,-176.003,8.363,148.488
C04436=1194.185,374.676,-78.793,-176.001,8.367,148.488
C04437=1194.181,374.924,-78.827,-176.000,8.369,148.489
C04438=1194.177,375.171,-78.862,-175.999,8.373,148.489
C04439=1194.173,375.419,-78.896,-175.997,8.376,148.490
C04440=1194.168,375.666,-78.931,-175.996,8.379,148.490
C04441=1194.165,375.914,-78.965,-175.995,8.382,148.491
C04442=1194.160,376.161,-78.999,-175.994,8.386,148.491
C04443=1194.157,376.409,-79.034,-175.993,8.389,148.492
C04444=1194.153,376.657,-79.068,-175.992,8.392,148.492
C04445=1194.149,376.905,-79.103,-175.990,8.394,148.492
C04446=1194.145,377.152,-79.137,-175.989,8.398,148.493
C04447=1194.140,377.399,-79.171,-175.988,8.401,148.493
C04448=1194.136,377.647,-79.206,-175.987,8.404,148.494
C04449=1194.132,377.895,-79.240,-175.986,8.407,148.494
C04450=1194.129,378.143,-79.275,-175.985,8.410,148.495
C04451=1194.124,378.390,-79.309,-175.983,8.414,148.495
C04452=1194.121,378.638,-79.343,-175.982,8.417,148.496
C04453=1194.116,378.885,-79.378,-175.981,8.420,148.496
C04454=1194.112,379.132,-79.413,-175.980,8.423,148.497
C04455=1194.109,379.380,-79.447,-175.980,8.426,148.498
C04456=1194.104,379.627,-79.482,-175.978,8.429,148.498
C04457=1194.100,379.876,-79.517,-175.977,8.433,148.499
C04458=1194.096,380.123,-79.550,-175.976,8.435,148.499
C04459=1194.092,380.371,-79.585,-175.975,8.438,148.500
C04460=1194.088,380.618,-79.620,-175.974,8.442,148.500
C04461=1194.084,380.866,-79.654,-175.973,8.444,148.501
C04462=1194.080,381.113,-79.689,-175.972,8.447,148.501
C04463=1194.076,381.361,-79.724,-175.971,8.451,148.502
C04464=1194.072,381.608,-79.759,-175.970,8.453,148.502
C04465=1194.068,381.856,-79.793,-175.969,8.456,148.503
C04466=1194.064,382.104,-79.827,-175.969,8.460,148.503
C04467=1194.060,382.351,-79.863,-175.967,8.462,148.504
C04468=1194.056,382.598,-79.897,-175.967,8.465,148.504
C04469=1194.052,382.846,-79.931,-175.966,8.469,148.505
C04470=1194.048,383.094,-79.966,-175.965,8.472,148.505
C04471=1194.044,383.342,-80.001,-175.964,8.474,148.506
C04472=1194.040,383.589,-80.036,-175.963,8.478,148.506
C04473=1194.036,383.836,-80.070,-175.962,8.481,148.507
C04474=1194.032,384.084,-80.105,-175.961,8.484,148.508
C04475=1194.028,384.331,-80.140,-175.961,8.487,148.508
C04476=1194.024,384.579,-80.175,-175.959,8.490,148.509
C04477=1194.020,384.827,-80.209,-175.959,8.493,148.509
C04478=1194.016,385.074,-80.243,-175.958,8.496,148.510
C04479=1194.012,385.321,-80.279,-175.958,8.498,148.510
C04480=1194.008,385.569,-80.313,-175.957,8.501,148.511
C04481=1194.004,385.817,-80.348,-175.956,8.504,148.511
C04482=1193.999,386.064,-80.383,-175.955,8.507,148.512
C04483=1193.996,386.312,-80.418,-175.954,8.510,148.512
C04484=1193.992,386.559,-80.452,-175.953,8.513,148.513
C04485=1193.988,386.807,-80.488,-175.953,8.516,148.514
C04486=1193.984,387.055,-80.522,-175.952,8.519,148.514
C04487=1193.979,387.302,-80.557,-175.951,8.522,148.515
C04488=1193.976,387.550,-80.592,-175.951,8.525,148.515
C04489=1193.972,387.797,-80.626,-175.950,8.527,148.516
C04490=1193.968,388.044,-80.662,-175.950,8.530,148.516
C04491=1193.964,388.292,-80.696,-175.949,8.533,148.517
C04492=1193.960,388.540,-80.731,-175.948,8.536,148.518
C04493=1193.956,388.787,-80.767,-175.948,8.539,148.518
C04494=1193.951,389.035,-80.801,-175.947,8.542,148.519
C04495=1193.948,389.282,-80.837,-175.946,8.545,148.519
C04496=1193.943,389.530,-80.871,-175.946,8.547,148.520
C04497=1193.940,389.777,-80.906,-175.945,8.550,148.520
C04498=1193.936,390.024,-80.941,-175.945,8.553,148.521
C04499=1193.932,390.272,-80.975,-175.944,8.556,148.522
C04500=1193.928,390.520,-81.011,-175.943,8.559,148.522
C04501=1193.923,390.767,-81.045,-175.943,8.561,148.523
C04502=1193.920,391.015,-81.081,-175.942,8.564,148.523
C04503=1193.915,391.262,-81.116,-175.942,8.566,148.524
C04504=1193.912,391.510,-81.151,-175.941,8.570,148.524
C04505=1193.908,391.758,-81.186,-175.941,8.572,148.525
C04506=1193.903,392.040,-81.226,-175.940,8.575,148.525
C04507=1193.899,392.324,-81.266,-175.939,8.578,148.526
C04508=1193.894,392.607,-81.306,-175.939,8.581,148.527
C04509=1193.890,392.890,-81.346,-175.938,8.584,148.527
C04510=1193.885,393.137,-81.381,-175.938,8.587,148.528
C04511=1193.881,393.385,-81.416,-175.937,8.590,148.529
C04512=1193.878,393.633,-81.451,-175.937,8.592,148.529
C04513=1193.873,393.880,-81.486,-175.936,8.595,148.530
C04514=1193.869,394.128,-81.521,-175.936,8.597,148.530
C04515=1193.866,394.375,-81.557,-175.935,8.601,148.531
C04516=1193.861,394.623,-81.591,-175.935,8.603,148.532
C04517=1193.858,394.870,-81.627,-175.935,8.605,148.532
C04518=1193.853,395.118,-81.661,-175.934,8.609,148.533
C04519=1193.849,395.365,-81.697,-175.934,8.611,148.533
C04520=1193.846,395.613,-81.732,-175.933,8.614,148.534
C04521=1193.841,395.860,-81.767,-175.933,8.616,148.534
C04522=1193.837,396.108,-81.802,-175.933,8.618,148.535
C04523=1193.833,396.356,-81.837,-175.932,8.622,148.535
C04524=1193.829,396.603,-81.872,-175.932,8.624,148.536
C04525=1193.826,396.850,-81.908,-175.932,8.626,148.536
C04526=1193.822,397.098,-81.943,-175.931,8.629,148.537
C04527=1193.817,397.345,-81.978,-175.931,8.632,148.538
C04528=1193.813,397.593,-82.013,-175.931,8.634,148.538
C04529=1193.809,397.840,-82.048,-175.931,8.636,148.539
C04530=1193.805,398.087,-82.084,-175.930,8.639,148.539
C04531=1193.801,398.335,-82.118,-175.929,8.642,148.540
C04532=1193.797,398.582,-82.154,-175.929,8.644,148.540
C04533=1193.794,398.830,-82.189,-175.929,8.646,148.541
C04534=1193.790,399.078,-82.224,-175.928,8.649,148.542
C04535=1193.785,399.325,-82.259,-175.928,8.652,148.542
C04536=1193.782,399.572,-82.295,-175.928,8.654,148.543
C04537=1193.778,399.820,-82.329,-175.928,8.656,148.543
C04538=1193.773,400.067,-82.365,-175.928,8.659,148.544
C04539=1193.770,400.315,-82.400,-175.927,8.662,148.544
C04540=1193.766,400.562,-82.436,-175.927,8.664,148.545
C04541=1193.762,400.810,-82.470,-175.926,8.666,148.546
C04542=1193.758,401.057,-82.506,-175.926,8.669,148.546
C04543=1193.754,401.305,-82.541,-175.926,8.671,148.547
C04544=1193.750,401.552,-82.576,-175.926,8.673,148.547
C04545=1193.746,401.799,-82.611,-175.925,8.675,148.548
C04546=1193.742,402.047,-82.647,-175.925,8.679,148.548
C04547=1193.738,402.295,-82.683,-175.925,8.681,148.549
C04548=1193.733,402.542,-82.717,-175.925,8.683,148.549
C04549=1193.730,402.790,-82.753,-175.924,8.686,148.550
C04550=1193.726,403.037,-82.789,-175.924,8.688,148.551
C04551=1193.722,403.284,-82.824,-175.924,8.690,148.551
C04552=1193.718,403.532,-82.859,-175.924,8.692,148.552
C04553=1193.714,403.780,-82.894,-175.923,8.695,148.552
C04554=1193.710,404.026,-82.929,-175.923,8.697,148.553
C04555=1193.706,404.274,-82.965,-175.923,8.699,148.553
C04556=1193.703,404.521,-83.000,-175.923,8.702,148.554
C04557=1193.698,404.770,-83.036,-175.923,8.704,148.554
C04558=1193.694,405.017,-83.071,-175.923,8.706,148.555
C04559=1193.690,405.264,-83.107,-175.922,8.708,148.555
C04560=1193.686,405.512,-83.142,-175.922,8.711,148.556
C04561=1193.682,405.758,-83.177,-175.922,8.713,148.557
C04562=1193.678,406.007,-83.212,-175.922,8.715,148.557
C04563=1193.674,406.254,-83.248,-175.921,8.718,148.558
C04564=1193.671,406.502,-83.283,-175.921,8.720,148.558
C04565=1193.666,406.749,-83.319,-175.921,8.722,148.559
C04566=1193.662,406.996,-83.355,-175.921,8.724,148.559
C04567=1193.658,407.244,-83.390,-175.920,8.727,148.560
C04568=1193.654,407.491,-83.425,-175.920,8.729,148.560
C04569=1193.650,407.739,-83.460,-175.920,8.731,148.561
C04570=1193.646,407.986,-83.496,-175.920,8.733,148.561
C04571=1193.643,408.234,-83.531,-175.920,8.736,148.562
C04572=1193.639,408.480,-83.566,-175.920,8.738,148.563
C04573=1193.634,408.728,-83.603,-175.919,8.741,148.563
C04574=1193.630,408.976,-83.638,-175.919,8.743,148.564
C04575=1193.626,409.224,-83.673,-175.920,8.744,148.564
C04576=1193.622,409.471,-83.708,-175.919,8.746,148.565
C04577=1193.619,409.718,-83.744,-175.919,8.749,148.565
C04578=1193.615,409.966,-83.779,-175.919,8.751,148.566
C04579=1193.610,410.213,-83.815,-175.919,8.753,148.566
C04580=1193.606,410.460,-83.851,-175.918,8.756,148.567
C04581=1193.603,410.708,-83.886,-175.918,8.758,148.567
C04582=1193.599,410.955,-83.922,-175.918,8.759,148.568
C04583=1193.595,411.203,-83.957,-175.918,8.762,148.568
C04584=1193.591,411.450,-83.992,-175.918,8.764,148.569
C04585=1193.586,411.698,-84.028,-175.918,8.766,148.569
C04586=1193.583,411.945,-84.063,-175.917,8.768,148.570
C04587=1193.579,412.193,-84.099,-175.917,8.771,148.570
C04588=1193.575,412.440,-84.134,-175.917,8.772,148.571
C04589=1193.571,412.687,-84.170,-175.917,8.774,148.571
C04590=1193.567,412.935,-84.206,-175.917,8.777,148.572
C04591=1193.563,413.183,-84.241,-175.917,8.779,148.572
C04592=1193.559,413.429,-84.276,-175.916,8.781,148.573
C04593=1193.555,413.677,-84.312,-175.917,8.783,148.573
C04594=1193.551,413.924,-84.348,-175.917,8.785,148.574
C04595=1193.547,414.172,-84.384,-175.916,8.787,148.574
C04596=1193.543,414.419,-84.419,-175.916,8.789,148.575
C04597=1193.539,414.666,-84.454,-175.915,8.791,148.575
C04598=1193.535,414.914,-84.490,-175.916,8.793,148.576
C04599=1193.531,415.162,-84.526,-175.915,8.795,148.576
C04600=1193.527,415.409,-84.562,-175.915,8.797,148.577
C04601=1193.523,415.656,-84.597,-175.915,8.799,148.577
C04602=1193.518,416.020,-84.649,-175.915,8.802,148.578
C04603=1193.513,416.385,-84.702,-175.915,8.805,148.579
C04604=1193.513,416.749,-84.753,-175.915,8.808,148.579
C04605=1193.516,417.112,-84.805,-175.914,8.811,148.580
C04606=1193.094,417.113,-84.845,-175.917,8.822,148.584
C04607=1193.091,416.746,-84.793,-175.918,8.818,148.583
C04608=1193.091,416.380,-84.741,-175.918,8.816,148.582
C04609=1193.095,416.013,-84.688,-175.918,8.813,148.582
C04610=1193.101,415.646,-84.635,-175.918,8.810,148.581
C04611=1193.105,415.398,-84.599,-175.918,8.808,148.580
C04612=1193.110,415.150,-84.563,-175.919,8.806,148.580
C04613=1193.114,414.904,-84.528,-175.919,8.803,148.579
C04614=1193.117,414.656,-84.492,-175.918,8.802,148.579
C04615=1193.121,414.409,-84.457,-175.919,8.800,148.578
C04616=1193.125,414.161,-84.421,-175.919,8.798,148.578
C04617=1193.130,413.913,-84.386,-175.920,8.795,148.578
C04618=1193.134,413.666,-84.351,-175.919,8.794,148.577
C04619=1193.137,413.418,-84.315,-175.920,8.792,148.577
C04620=1193.141,413.171,-84.280,-175.920,8.789,148.576
C04621=1193.146,412.924,-84.244,-175.920,8.787,148.575
C04622=1193.150,412.676,-84.208,-175.920,8.785,148.575
C04623=1193.153,412.429,-84.173,-175.920,8.783,148.574
C04624=1193.157,412.181,-84.137,-175.920,8.781,148.574
C04625=1193.161,411.934,-84.102,-175.921,8.779,148.573
C04626=1193.166,411.687,-84.066,-175.921,8.777,148.573
C04627=1193.169,411.439,-84.030,-175.921,8.774,148.572
C04628=1193.173,411.192,-83.995,-175.921,8.772,148.572
C04629=1193.177,410.944,-83.959,-175.921,8.771,148.571
C04630=1193.181,410.697,-83.924,-175.921,8.768,148.571
C04631=1193.185,410.450,-83.888,-175.921,8.766,148.570
C04632=1193.189,410.202,-83.852,-175.922,8.764,148.570
C04633=1193.193,409.955,-83.817,-175.922,8.762,148.569
C04634=1193.197,409.707,-83.782,-175.922,8.759,148.569
C04635=1193.201,409.460,-83.747,-175.922,8.757,148.568
C04636=1193.205,409.212,-83.711,-175.922,8.755,148.568
C04637=1193.209,408.964,-83.675,-175.922,8.753,148.567
C04638=1193.213,408.718,-83.640,-175.922,8.751,148.567
C04639=1193.217,408.470,-83.604,-175.922,8.749,148.566
C04640=1193.221,408.223,-83.569,-175.923,8.746,148.565
C04641=1193.224,407.975,-83.533,-175.923,8.744,148.565
C04642=1193.229,407.728,-83.499,-175.923,8.742,148.564
C04643=1193.232,407.480,-83.463,-175.923,8.740,148.564
C04644=1193.237,407.232,-83.427,-175.924,8.737,148.563
C04645=1193.241,406.986,-83.392,-175.924,8.735,148.563
C04646=1193.245,406.738,-83.356,-175.924,8.733,148.562
C04647=1193.248,406.491,-83.321,-175.924,8.730,148.562
C04648=1193.252,406.243,-83.285,-175.924,8.729,148.561
C04649=1193.257,405.996,-83.251,-175.924,8.727,148.561
C04650=1193.260,405.748,-83.215,-175.924,8.725,148.560
C04651=1193.265,405.500,-83.179,-175.924,8.722,148.560
C04652=1193.268,405.253,-83.144,-175.925,8.720,148.559
C04653=1193.273,405.006,-83.108,-175.925,8.717,148.558
C04654=1193.276,404.758,-83.073,-175.925,8.715,148.558
C04655=1193.280,404.510,-83.038,-175.925,8.713,148.557
C04656=1193.285,404.264,-83.003,-175.926,8.711,148.557
C04657=1193.288,404.016,-82.967,-175.926,8.708,148.556
C04658=1193.292,403.769,-82.932,-175.927,8.705,148.556
C04659=1193.296,403.521,-82.897,-175.927,8.703,148.555
C04660=1193.301,403.273,-82.861,-175.927,8.701,148.555
C04661=1193.305,403.026,-82.826,-175.927,8.698,148.554
C04662=1193.308,402.778,-82.790,-175.927,8.696,148.553
C04663=1193.312,402.532,-82.755,-175.927,8.694,148.553
C04664=1193.316,402.283,-82.720,-175.928,8.691,148.552
C04665=1193.320,402.036,-82.685,-175.928,8.689,148.552
C04666=1193.324,401.789,-82.649,-175.928,8.687,148.551
C04667=1193.328,401.542,-82.614,-175.928,8.685,148.551
C04668=1193.332,401.293,-82.579,-175.929,8.682,148.550
C04669=1193.336,401.047,-82.544,-175.929,8.679,148.550
C04670=1193.340,400.799,-82.508,-175.929,8.677,148.549
C04671=1193.344,400.552,-82.473,-175.929,8.674,148.548
C04672=1193.348,400.304,-82.438,-175.930,8.672,148.548
C04673=1193.353,400.056,-82.402,-175.930,8.670,148.547
C04674=1193.356,399.809,-82.367,-175.930,8.668,148.547
C04675=1193.361,399.562,-82.332,-175.931,8.664,148.546
C04676=1193.364,399.314,-82.297,-175.931,8.662,148.546
C04677=1193.368,399.067,-82.261,-175.931,8.660,148.545
C04678=1193.373,398.819,-82.227,-175.932,8.658,148.545
C04679=1193.376,398.572,-82.191,-175.931,8.655,148.544
C04680=1193.380,398.324,-82.155,-175.932,8.652,148.543
C04681=1193.385,398.077,-82.121,-175.932,8.650,148.543
C04682=1193.388,397.829,-82.085,-175.933,8.647,148.542
C04683=1193.392,397.582,-82.050,-175.933,8.645,148.542
C04684=1193.396,397.334,-82.015,-175.934,8.642,148.541
C04685=1193.400,397.087,-81.980,-175.934,8.640,148.541
C04686=1193.404,396.839,-81.944,-175.934,8.638,148.540
C04687=1193.408,396.592,-81.910,-175.935,8.634,148.539
C04688=1193.412,396.344,-81.874,-175.935,8.632,148.539
C04689=1193.416,396.097,-81.839,-175.935,8.630,148.538
C04690=1193.420,395.849,-81.804,-175.936,8.627,148.538
C04691=1193.424,395.602,-81.769,-175.936,8.624,148.537
C04692=1193.428,395.354,-81.734,-175.936,8.622,148.537
C04693=1193.432,395.107,-81.699,-175.937,8.619,148.536
C04694=1193.436,394.860,-81.663,-175.937,8.617,148.536
C04695=1193.440,394.612,-81.629,-175.938,8.614,148.535
C04696=1193.444,394.365,-81.593,-175.938,8.611,148.534
C04697=1193.448,394.116,-81.558,-175.938,8.609,148.534
C04698=1193.452,393.870,-81.523,-175.939,8.606,148.533
C04699=1193.456,393.622,-81.488,-175.939,8.603,148.533
C04700=1193.460,393.374,-81.453,-175.940,8.600,148.532
C04701=1193.464,393.127,-81.418,-175.940,8.598,148.531
C04702=1193.468,392.879,-81.383,-175.941,8.595,148.531
C04703=1193.472,392.597,-81.343,-175.941,8.593,148.530
C04704=1193.477,392.313,-81.303,-175.942,8.589,148.530
C04705=1193.482,392.029,-81.262,-175.942,8.586,148.529
C04706=1193.486,391.746,-81.223,-175.943,8.583,148.528
C04707=1193.490,391.499,-81.187,-175.944,8.580,148.528
C04708=1193.494,391.252,-81.153,-175.944,8.578,148.527
C04709=1193.498,391.004,-81.117,-175.945,8.574,148.527
C04710=1193.502,390.756,-81.083,-175.945,8.572,148.526
C04711=1193.506,390.509,-81.047,-175.946,8.569,148.525
C04712=1193.510,390.261,-81.013,-175.946,8.567,148.525
C04713=1193.515,390.014,-80.977,-175.947,8.563,148.524
C04714=1193.518,389.766,-80.943,-175.947,8.560,148.524
C04715=1193.522,389.518,-80.908,-175.948,8.558,148.523
C04716=1193.526,389.271,-80.873,-175.948,8.555,148.523
C04717=1193.530,389.023,-80.838,-175.949,8.552,148.522
C04718=1193.534,388.777,-80.803,-175.949,8.550,148.521
C04719=1193.538,388.528,-80.768,-175.950,8.547,148.521
C04720=1193.542,388.282,-80.733,-175.951,8.543,148.520
C04721=1193.546,388.033,-80.698,-175.951,8.541,148.520
C04722=1193.550,387.785,-80.663,-175.953,8.538,148.519
C04723=1193.554,387.539,-80.629,-175.953,8.535,148.519
C04724=1193.558,387.291,-80.594,-175.954,8.532,148.518
C04725=1193.562,387.044,-80.559,-175.954,8.530,148.518
C04726=1193.566,386.796,-80.524,-175.955,8.527,148.517
C04727=1193.571,386.548,-80.490,-175.956,8.524,148.516
C04728=1193.574,386.301,-80.454,-175.957,8.521,148.516
C04729=1193.578,386.054,-80.420,-175.957,8.518,148.515
C04730=1193.582,385.806,-80.385,-175.958,8.515,148.515
C04731=1193.586,385.558,-80.350,-175.959,8.512,148.514
C04732=1193.590,385.311,-80.315,-175.959,8.509,148.514
C04733=1193.594,385.063,-80.280,-175.961,8.506,148.513
C04734=1193.598,384.816,-80.246,-175.961,8.503,148.513
C04735=1193.602,384.568,-80.211,-175.962,8.500,148.512
C04736=1193.606,384.321,-80.177,-175.963,8.497,148.511
C04737=1193.610,384.073,-80.141,-175.963,8.495,148.511
C04738=1193.615,383.826,-80.107,-175.964,8.492,148.510
C04739=1193.618,383.578,-80.072,-175.965,8.489,148.510
C04740=1193.622,383.330,-80.038,-175.966,8.486,148.509
C04741=1193.626,383.083,-80.002,-175.967,8.483,148.509
C04742=1193.631,382.836,-79.968,-175.968,8.479,148.508
C04743=1193.635,382.587,-79.933,-175.969,8.477,148.508
C04744=1193.638,382.340,-79.899,-175.970,8.474,148.507
C04745=1193.642,382.093,-79.864,-175.970,8.470,148.507
C04746=1193.647,381.845,-79.829,-175.971,8.467,148.506
C04747=1193.651,381.597,-79.794,-175.972,8.465,148.506
C04748=1193.655,381.350,-79.760,-175.973,8.461,148.505
C04749=1193.658,381.102,-79.726,-175.974,8.458,148.504
C04750=1193.663,380.855,-79.690,-175.976,8.455,148.504
C04751=1193.666,380.607,-79.656,-175.977,8.452,148.503
C04752=1193.671,380.360,-79.622,-175.977,8.449,148.503
C04753=1193.675,380.112,-79.587,-175.979,8.446,148.502
C04754=1193.679,379.864,-79.552,-175.979,8.443,148.502
C04755=1193.682,379.617,-79.518,-175.981,8.440,148.502
C04756=1193.687,379.369,-79.484,-175.981,8.437,148.501
C04757=1193.691,379.122,-79.448,-175.982,8.434,148.500
C04758=1193.694,378.875,-79.414,-175.984,8.430,148.500
C04759=1193.699,378.627,-79.380,-175.985,8.427,148.499
C04760=1193.703,378.379,-79.345,-175.986,8.424,148.499
C04761=1193.707,378.132,-79.311,-175.987,8.421,148.498
C04762=1193.711,377.884,-79.276,-175.988,8.418,148.498
C04763=1193.715,377.636,-79.242,-175.989,8.414,148.497
C04764=1193.719,377.389,-79.208,-175.991,8.411,148.497
C04765=1193.723,377.141,-79.173,-175.991,8.408,148.496
C04766=1193.727,376.893,-79.138,-175.993,8.406,148.496
C04767=1193.731,376.646,-79.104,-175.994,8.402,148.495
C04768=1193.735,376.399,-79.070,-175.995,8.399,148.495
C04769=1193.739,376.151,-79.036,-175.996,8.396,148.494
C04770=1193.743,375.903,-79.001,-175.997,8.393,148.494
C04771=1193.747,375.655,-78.966,-175.999,8.389,148.494
C04772=1193.751,375.408,-78.933,-176.000,8.386,148.493
C04773=1193.756,375.161,-78.898,-176.001,8.383,148.493
C04774=1193.759,374.913,-78.864,-176.002,8.379,148.492
C04775=1193.763,374.665,-78.829,-176.004,8.377,148.492
C04776=1193.767,374.417,-78.795,-176.005,8.374,148.491
C04777=1193.771,374.170,-78.761,-176.006,8.370,148.490
C04778=1193.776,373.923,-78.726,-176.007,8.367,148.490
C04779=1193.779,373.675,-78.692,-176.009,8.364,148.490
C04780=1193.784,373.428,-78.657,-176.011,8.361,148.489
C04781=1193.787,373.180,-78.623,-176.011,8.358,148.489
C04782=1193.792,372.932,-78.589,-176.013,8.354,148.488
C04783=1193.796,372.685,-78.556,-176.014,8.351,148.488
C04784=1193.800,372.436,-78.521,-176.016,8.348,148.487
C04785=1193.803,372.189,-78.487,-176.017,8.344,148.487
C04786=1193.808,371.942,-78.452,-176.018,8.342,148.486
C04787=1193.811,371.694,-78.418,-176.020,8.338,148.486
C04788=1193.816,371.447,-78.384,-176.021,8.335,148.486
C04789=1193.820,371.199,-78.351,-176.023,8.332,148.485
C04790=1193.824,370.951,-78.316,-176.024,8.328,148.485
C04791=1193.828,370.704,-78.282,-176.025,8.326,148.484
C04792=1193.832,370.456,-78.247,-176.027,8.322,148.484
C04793=1193.836,370.208,-78.214,-176.028,8.319,148.483
C04794=1193.840,369.960,-78.179,-176.030,8.316,148.483
C04795=1193.844,369.713,-78.146,-176.031,8.313,148.483
C04796=1193.848,369.465,-78.111,-176.033,8.309,148.482
C04797=1193.852,369.218,-78.078,-176.034,8.306,148.482
C04798=1193.857,368.970,-78.043,-176.036,8.303,148.481
C04799=1193.860,368.722,-78.009,-176.037,8.300,148.481
C04800=1193.864,368.475,-77.975,-176.039,8.296,148.480
C04801=1193.869,368.227,-77.941,-176.041,8.293,148.480
C04802=1193.872,367.979,-77.907,-176.042,8.290,148.480
C04803=1193.877,367.732,-77.873,-176.044,8.286,148.479
C04804=1193.881,367.484,-77.839,-176.045,8.283,148.479
C04805=1193.884,367.236,-77.805,-176.047,8.280,148.478
C04806=1193.889,366.988,-77.771,-176.048,8.277,148.478
C04807=1193.894,366.708,-77.733,-176.050,8.273,148.478
C04808=1193.898,366.427,-77.694,-176.052,8.269,148.477
C04809=1193.902,366.146,-77.656,-176.054,8.265,148.477
C04810=1193.907,365.865,-77.617,-176.056,8.262,148.476
C04811=1193.911,365.617,-77.584,-176.057,8.259,148.476
C04812=1193.915,365.370,-77.550,-176.059,8.255,148.475
C04813=1193.919,365.122,-77.516,-176.060,8.252,148.475
C04814=1193.923,364.875,-77.482,-176.062,8.249,148.475
C04815=1193.927,364.627,-77.449,-176.064,8.245,148.474
C04816=1193.931,364.379,-77.414,-176.066,8.242,148.474
C04817=1193.935,364.131,-77.381,-176.067,8.239,148.474
C04818=1193.939,363.884,-77.347,-176.069,8.235,148.473
C04819=1193.944,363.636,-77.313,-176.070,8.232,148.473
C04820=1193.947,363.388,-77.279,-176.072,8.229,148.472
C04821=1193.952,363.140,-77.246,-176.074,8.226,148.472
C04822=1193.955,362.893,-77.212,-176.076,8.222,148.472
C04823=1193.960,362.645,-77.178,-176.077,8.220,148.471
C04824=1193.964,362.397,-77.144,-176.079,8.216,148.471
C04825=1193.968,362.150,-77.111,-176.081,8.212,148.471
C04826=1193.972,361.902,-77.078,-176.082,8.209,148.470
C04827=1193.976,361.655,-77.044,-176.084,8.206,148.470
C04828=1193.980,361.407,-77.010,-176.086,8.202,148.470
C04829=1193.984,361.159,-76.976,-176.088,8.200,148.469
C04830=1193.988,360.911,-76.943,-176.090,8.196,148.469
C04831=1193.992,360.663,-76.910,-176.091,8.193,148.468
C04832=1193.996,360.416,-76.876,-176.094,8.189,148.468
C04833=1194.001,360.168,-76.842,-176.095,8.187,148.468
C04834=1194.005,359.921,-76.809,-176.097,8.183,148.468
C04835=1194.008,359.672,-76.775,-176.099,8.180,148.467
C04836=1194.012,359.425,-76.741,-176.101,8.176,148.467
C04837=1194.016,359.177,-76.708,-176.102,8.173,148.467
C04838=1194.020,358.930,-76.675,-176.104,8.170,148.466
C04839=1194.025,358.682,-76.641,-176.106,8.167,148.466
C04840=1194.029,358.434,-76.607,-176.108,8.163,148.465
C04841=1194.033,358.187,-76.574,-176.111,8.160,148.465
C04842=1194.037,357.938,-76.541,-176.112,8.157,148.465
C04843=1194.041,357.690,-76.508,-176.114,8.153,148.465
C04844=1194.045,357.443,-76.474,-176.116,8.150,148.464
C04845=1194.049,357.196,-76.441,-176.118,8.146,148.464
C04846=1194.053,356.948,-76.407,-176.120,8.144,148.464
C04847=1194.057,356.700,-76.374,-176.121,8.140,148.463
C04848=1194.062,356.452,-76.341,-176.124,8.137,148.463
C04849=1194.066,356.204,-76.307,-176.126,8.134,148.463
C04850=1194.070,355.957,-76.273,-176.128,8.130,148.462
C04851=1194.074,355.709,-76.240,-176.129,8.128,148.462
C04852=1194.078,355.461,-76.207,-176.132,8.124,148.462
C04853=1194.082,355.213,-76.174,-176.133,8.121,148.462
C04854=1194.086,354.966,-76.140,-176.136,8.117,148.461
C04855=1194.090,354.718,-76.107,-176.138,8.114,148.461
C04856=1194.094,354.470,-76.074,-176.139,8.111,148.461
C04857=1194.098,354.223,-76.041,-176.141,8.108,148.461
C04858=1194.103,353.975,-76.008,-176.144,8.104,148.460
C04859=1194.107,353.727,-75.975,-176.145,8.101,148.460
C04860=1194.111,353.479,-75.942,-176.148,8.097,148.460
C04861=1194.115,353.232,-75.908,-176.149,8.095,148.460
C04862=1194.119,352.984,-75.875,-176.152,8.092,148.459
C04863=1194.123,352.736,-75.842,-176.153,8.088,148.459
C04864=1194.127,352.488,-75.809,-176.156,8.085,148.459
C04865=1194.132,352.241,-75.776,-176.157,8.082,148.458
C04866=1194.136,351.993,-75.743,-176.159,8.079,148.458
C04867=1194.140,351.745,-75.709,-176.161,8.075,148.458
C04868=1194.143,351.498,-75.677,-176.163,8.072,148.458
C04869=1194.148,351.249,-75.644,-176.166,8.069,148.457
C04870=1194.152,351.002,-75.611,-176.167,8.066,148.457
C04871=1194.156,350.754,-75.578,-176.170,8.063,148.457
C04872=1194.160,350.506,-75.545,-176.171,8.059,148.457
C04873=1194.164,350.259,-75.512,-176.174,8.056,148.456
C04874=1194.168,350.011,-75.479,-176.176,8.052,148.456
C04875=1194.173,349.763,-75.446,-176.178,8.050,148.456
C04876=1194.177,349.515,-75.413,-176.180,8.047,148.456
C04877=1194.180,349.267,-75.381,-176.182,8.043,148.455
C04878=1194.185,349.020,-75.347,-176.184,8.040,148.455
C04879=1194.189,348.772,-75.314,-176.187,8.037,148.455
C04880=1194.193,348.523,-75.282,-176.188,8.034,148.455
C04881=1194.197,348.276,-75.249,-176.190,8.031,148.454
C04882=1194.201,348.028,-75.215,-176.192,8.027,148.454
C04883=1194.205,347.781,-75.183,-176.194,8.024,148.454
C04884=1194.209,347.532,-75.150,-176.197,8.021,148.454
C04885=1194.213,347.285,-75.117,-176.198,8.018,148.454
C04886=1194.217,347.037,-75.084,-176.201,8.015,148.453
C04887=1194.222,346.788,-75.052,-176.203,8.011,148.453
C04888=1194.226,346.542,-75.020,-176.205,8.008,148.453
C04889=1194.230,346.294,-74.986,-176.207,8.005,148.453
C04890=1194.235,346.046,-74.954,-176.209,8.002,148.453
C04891=1194.239,345.798,-74.921,-176.211,7.999,148.452
C04892=1194.242,345.551,-74.888,-176.213,7.996,148.452
C04893=1194.246,345.302,-74.856,-176.216,7.992,148.452
C04894=1194.251,345.054,-74.823,-176.218,7.989,148.452
C04895=1194.255,344.806,-74.790,-176.220,7.986,148.451
C04896=1194.258,344.559,-74.758,-176.222,7.983,148.451
C04897=1194.264,344.311,-74.726,-176.224,7.980,148.451
C04898=1194.268,344.063,-74.692,-176.226,7.976,148.451
C04899=1194.272,343.815,-74.660,-176.229,7.973,148.451
C04900=1194.276,343.568,-74.627,-176.230,7.971,148.450
C04901=1194.280,343.319,-74.595,-176.232,7.967,148.450
C04902=1194.284,343.071,-74.562,-176.235,7.964,148.450
C04903=1194.288,342.823,-74.530,-176.237,7.961,148.450
C04904=1194.293,342.576,-74.497,-176.239,7.957,148.450
C04905=1194.297,342.328,-74.465,-176.242,7.954,148.449
C04906=1194.300,342.081,-74.432,-176.244,7.952,148.449
C04907=1194.305,341.832,-74.400,-176.246,7.948,148.449
C04908=1194.308,341.585,-74.367,-176.248,7.945,148.449
C04909=1194.313,341.336,-74.335,-176.250,7.942,148.449
C04910=1194.318,341.089,-74.303,-176.253,7.938,148.448
C04911=1194.322,340.810,-74.266,-176.255,7.935,148.448
C04912=1194.327,340.532,-74.229,-176.257,7.932,148.448
C04913=1194.331,340.253,-74.193,-176.260,7.929,148.448
C04914=1194.336,339.974,-74.157,-176.262,7.925,148.448
C04915=1194.340,339.727,-74.125,-176.264,7.922,148.448
C04916=1194.344,339.479,-74.092,-176.266,7.919,148.447
C04917=1194.349,339.231,-74.060,-176.269,7.915,148.447
C04918=1194.352,338.983,-74.027,-176.271,7.912,148.447
C04919=1194.357,338.735,-73.995,-176.274,7.909,148.447
C04920=1194.361,338.487,-73.964,-176.275,7.907,148.447
C04921=1194.365,338.239,-73.931,-176.277,7.903,148.447
C04922=1194.369,337.992,-73.899,-176.280,7.900,148.446
C04923=1194.373,337.743,-73.866,-176.282,7.897,148.446
C04924=1194.377,337.496,-73.835,-176.285,7.894,148.446
C04925=1194.382,337.248,-73.802,-176.286,7.891,148.446
C04926=1194.386,337.000,-73.770,-176.289,7.888,148.446
C04927=1194.389,336.752,-73.738,-176.291,7.885,148.446
C04928=1194.394,336.505,-73.706,-176.293,7.881,148.445
C04929=1194.398,336.257,-73.674,-176.296,7.878,148.445
C04930=1194.402,336.008,-73.641,-176.297,7.876,148.445
C04931=1194.407,335.761,-73.610,-176.300,7.873,148.445
C04932=1194.411,335.512,-73.577,-176.302,7.869,148.445
C04933=1194.415,335.264,-73.546,-176.305,7.866,148.445
C04934=1194.418,335.016,-73.514,-176.307,7.863,148.445
C04935=1194.423,334.769,-73.481,-176.309,7.860,148.444
C04936=1194.427,334.521,-73.449,-176.311,7.857,148.444
C04937=1194.431,334.273,-73.417,-176.314,7.854,148.444
C04938=1194.436,334.026,-73.385,-176.316,7.851,148.444
C04939=1194.439,333.778,-73.353,-176.318,7.847,148.444
C04940=1194.444,333.529,-73.321,-176.320,7.845,148.444
C04941=1194.448,333.282,-73.289,-176.323,7.842,148.444
C04942=1194.452,333.034,-73.258,-176.325,7.839,148.443
C04943=1194.456,332.786,-73.225,-176.328,7.835,148.443
C04944=1194.461,332.538,-73.194,-176.330,7.832,148.443
C04945=1194.464,332.290,-73.162,-176.332,7.830,148.443
C04946=1194.469,332.041,-73.130,-176.334,7.827,148.443
C04947=1194.473,331.794,-73.099,-176.336,7.823,148.443
C04948=1194.477,331.546,-73.067,-176.339,7.820,148.443
C04949=1194.481,331.297,-73.034,-176.341,7.817,148.443
C04950=1194.486,331.050,-73.003,-176.343,7.814,148.442
C04951=1194.489,330.802,-72.971,-176.346,7.811,148.442
C04952=1194.494,330.555,-72.940,-176.348,7.808,148.442
C04953=1194.498,330.306,-72.907,-176.351,7.805,148.442
C04954=1194.502,330.058,-72.876,-176.353,7.802,148.442
C04955=1194.507,329.810,-72.845,-176.355,7.799,148.442
C04956=1194.510,329.562,-72.813,-176.357,7.796,148.442
C04957=1194.515,329.315,-72.781,-176.360,7.793,148.442
C04958=1194.519,329.067,-72.749,-176.362,7.790,148.442
C04959=1194.523,328.818,-72.718,-176.364,7.787,148.441
C04960=1194.527,328.571,-72.686,-176.367,7.784,148.441
C04961=1194.532,328.322,-72.654,-176.369,7.781,148.441
C04962=1194.536,328.075,-72.622,-176.372,7.778,148.441
C04963=1194.540,327.826,-72.591,-176.374,7.775,148.441
C04964=1194.544,327.579,-72.560,-176.375,7.772,148.441
C04965=1194.548,327.331,-72.528,-176.378,7.769,148.441
C04966=1194.552,327.082,-72.497,-176.380,7.766,148.441
C04967=1194.557,326.835,-72.465,-176.383,7.763,148.441
C04968=1194.561,326.587,-72.433,-176.385,7.760,148.440
C04969=1194.565,326.339,-72.402,-176.387,7.757,148.441
C04970=1194.569,326.091,-72.370,-176.390,7.754,148.440
C04971=1194.573,325.843,-72.339,-176.392,7.751,148.440
C04972=1194.577,325.595,-72.307,-176.395,7.748,148.440
C04973=1194.582,325.347,-72.276,-176.397,7.745,148.440
C04974=1194.586,325.099,-72.245,-176.399,7.742,148.440
C04975=1194.590,324.851,-72.213,-176.402,7.739,148.440
C04976=1194.594,324.603,-72.182,-176.404,7.736,148.440
C04977=1194.598,324.355,-72.151,-176.407,7.733,148.440
C04978=1194.602,324.107,-72.119,-176.409,7.731,148.440
C04979=1194.607,323.859,-72.088,-176.411,7.727,148.440
C04980=1194.611,323.611,-72.056,-176.414,7.724,148.440
C04981=1194.616,323.363,-72.025,-176.416,7.721,148.439
C04982=1194.619,323.115,-71.993,-176.419,7.718,148.439
C04983=1194.624,322.867,-71.962,-176.421,7.716,148.439
C04984=1194.628,322.619,-71.931,-176.423,7.712,148.439
C04985=1194.632,322.371,-71.900,-176.426,7.709,148.439
C04986=1194.636,322.122,-71.869,-176.428,7.706,148.439
C04987=1194.641,321.875,-71.837,-176.430,7.704,148.439
C04988=1194.645,321.626,-71.806,-176.432,7.701,148.439
C04989=1194.648,321.379,-71.775,-176.435,7.697,148.439
C04990=1194.653,321.131,-71.744,-176.438,7.694,148.439
C04991=1194.657,320.883,-71.713,-176.440,7.691,148.439
C04992=1194.661,320.635,-71.682,-176.442,7.689,148.439
C04993=1194.665,320.387,-71.651,-176.445,7.686,148.439
C04994=1194.670,320.139,-71.620,-176.447,7.683,148.438
C04995=1194.674,319.891,-71.588,-176.450,7.680,148.438
C04996=1194.678,319.643,-71.557,-176.451,7.677,148.438
C04997=1194.683,319.395,-71.526,-176.454,7.674,148.438
C04998=1194.687,319.147,-71.495,-176.457,7.671,148.438
C04999=1194.691,318.899,-71.464,-176.459,7.668,148.438
C05000=1194.695,318.650,-71.433,-176.462,7.665,148.438
C05001=1194.699,318.402,-71.403,-176.464,7.663,148.438
C05002=1194.703,318.155,-71.371,-176.466,7.659,148.438
C05003=1194.707,317.906,-71.340,-176.469,7.656,148.438
C05004=1194.712,317.659,-71.309,-176.471,7.653,148.438
C05005=1194.717,317.411,-71.278,-176.473,7.651,148.438
C05006=1194.721,317.162,-71.247,-176.476,7.648,148.438
C05007=1194.724,316.915,-71.216,-176.479,7.645,148.438
C05008=1194.729,316.667,-71.186,-176.481,7.641,148.438
C05009=1194.733,316.418,-71.155,-176.483,7.639,148.438
C05010=1194.737,316.170,-71.124,-176.486,7.636,148.438
C05011=1194.742,315.922,-71.093,-176.488,7.633,148.438
C05012=1194.745,315.674,-71.062,-176.491,7.630,148.437
C05013=1194.750,315.426,-71.032,-176.493,7.628,148.438
C05014=1194.755,315.178,-71.001,-176.495,7.625,148.438
C05015=1194.759,314.902,-70.966,-176.498,7.621,148.437
C05016=1194.763,314.626,-70.932,-176.501,7.617,148.437
C05017=1194.768,314.349,-70.898,-176.504,7.614,148.437
C05018=1194.773,314.073,-70.864,-176.506,7.611,148.437
C05019=1194.777,313.824,-70.833,-176.509,7.608,148.437
C05020=1194.781,313.576,-70.802,-176.511,7.606,148.437
C05021=1194.786,313.328,-70.771,-176.513,7.603,148.437
C05022=1194.790,313.081,-70.741,-176.516,7.600,148.437
C05023=1194.794,312.832,-70.710,-176.519,7.597,148.437
C05024=1194.798,312.584,-70.679,-176.520,7.594,148.437
C05025=1194.802,312.336,-70.649,-176.523,7.591,148.437
C05026=1194.807,312.088,-70.618,-176.526,7.588,148.437
C05027=1194.811,311.840,-70.587,-176.529,7.585,148.437
C05028=1194.815,311.592,-70.558,-176.530,7.583,148.437
C05029=1194.820,311.344,-70.527,-176.533,7.580,148.437
C05030=1194.824,311.096,-70.496,-176.536,7.577,148.437
C05031=1194.828,310.847,-70.466,-176.538,7.574,148.437
C05032=1194.832,310.599,-70.435,-176.540,7.572,148.437
C05033=1194.836,310.352,-70.405,-176.543,7.568,148.437
C05034=1194.841,310.104,-70.374,-176.545,7.565,148.437
C05035=1194.845,309.854,-70.343,-176.548,7.562,148.437
C05036=1194.849,309.607,-70.313,-176.550,7.560,148.437
C05037=1194.854,309.359,-70.282,-176.553,7.557,148.437
C05038=1194.857,309.111,-70.252,-176.555,7.554,148.437
C05039=1194.862,308.863,-70.222,-176.558,7.551,148.437
C05040=1194.867,308.615,-70.191,-176.560,7.548,148.437
C05041=1194.870,308.366,-70.161,-176.563,7.545,148.437
C05042=1194.875,308.118,-70.130,-176.565,7.542,148.437
C05043=1194.879,307.870,-70.101,-176.568,7.539,148.437
C05044=1194.884,307.622,-70.070,-176.570,7.537,148.437
C05045=1194.888,307.374,-70.040,-176.572,7.534,148.437
C05046=1194.892,307.126,-70.010,-176.575,7.531,148.437
C05047=1194.896,306.878,-69.979,-176.577,7.529,148.437
C05048=1194.900,306.630,-69.948,-176.580,7.526,148.437
C05049=1194.905,306.381,-69.919,-176.583,7.523,148.437
C05050=1194.909,306.133,-69.888,-176.585,7.519,148.437
C05051=1194.913,305.885,-69.859,-176.587,7.517,148.437
C05052=1194.918,305.637,-69.828,-176.590,7.514,148.437
C05053=1194.922,305.389,-69.798,-176.592,7.511,148.437
C05054=1194.926,305.140,-69.767,-176.595,7.509,148.437
C05055=1194.930,304.893,-69.737,-176.597,7.506,148.437
C05056=1194.934,304.644,-69.708,-176.600,7.503,148.437
C05057=1194.939,304.396,-69.677,-176.602,7.500,148.437
C05058=1194.943,304.148,-69.648,-176.604,7.497,148.437
C05059=1194.948,303.900,-69.617,-176.607,7.494,148.437
C05060=1194.952,303.652,-69.587,-176.610,7.491,148.437
C05061=1194.956,303.404,-69.557,-176.613,7.488,148.437
C05062=1194.961,303.156,-69.527,-176.615,7.486,148.437
C05063=1194.964,302.908,-69.497,-176.617,7.483,148.437
C05064=1194.969,302.659,-69.467,-176.620,7.480,148.437
C05065=1194.974,302.411,-69.437,-176.622,7.478,148.437
C05066=1194.977,302.163,-69.407,-176.625,7.475,148.437
C05067=1194.982,301.914,-69.377,-176.627,7.472,148.437
C05068=1194.986,301.667,-69.347,-176.629,7.469,148.437
C05069=1194.990,301.418,-69.317,-176.632,7.466,148.437
C05070=1194.995,301.170,-69.287,-176.635,7.463,148.437
C05071=1194.999,300.922,-69.257,-176.637,7.460,148.437
C05072=1195.003,300.674,-69.228,-176.640,7.458,148.437
C05073=1195.007,300.425,-69.198,-176.642,7.455,148.437
C05074=1195.012,300.178,-69.167,-176.645,7.452,148.437
C05075=1195.016,299.929,-69.138,-176.647,7.450,148.437
C05076=1195.020,299.681,-69.108,-176.650,7.447,148.437
C05077=1195.025,299.433,-69.078,-176.652,7.444,148.437
C05078=1195.029,299.185,-69.048,-176.655,7.442,148.437
C05079=1195.033,298.937,-69.019,-176.657,7.439,148.437
C05080=1195.037,298.688,-68.989,-176.660,7.436,148.437
C05081=1195.041,298.441,-68.959,-176.663,7.433,148.437
C05082=1195.046,298.192,-68.929,-176.665,7.431,148.437
C05083=1195.050,297.944,-68.900,-176.667,7.427,148.437
C05084=1195.054,297.695,-68.870,-176.670,7.424,148.437
C05085=1195.058,297.447,-68.841,-176.672,7.422,148.437
C05086=1195.063,297.199,-68.811,-176.675,7.419,148.437
C05087=1195.067,296.951,-68.781,-176.677,7.416,148.437
C05088=1195.071,296.703,-68.751,-176.680,7.414,148.437
C05089=1195.076,296.454,-68.722,-176.682,7.411,148.437
C05090=1195.080,296.206,-68.692,-176.685,7.408,148.437
C05091=1195.085,295.959,-68.663,-176.687,7.406,148.437
C05092=1195.089,295.710,-68.634,-176.690,7.403,148.437
C05093=1195.093,295.462,-68.604,-176.692,7.400,148.437
C05094=1195.097,295.214,-68.575,-176.695,7.397,148.437
C05095=1195.102,294.965,-68.545,-176.697,7.394,148.437
C05096=1195.106,294.717,-68.515,-176.700,7.391,148.437
C05097=1195.110,294.469,-68.486,-176.702,7.389,148.437
C05098=1195.115,294.220,-68.456,-176.705,7.386,148.438
C05099=1195.119,293.972,-68.427,-176.708,7.383,148.438
C05100=1195.123,293.724,-68.397,-176.710,7.381,148.438
C05101=1195.127,293.476,-68.368,-176.712,7.378,148.438
C05102=1195.131,293.227,-68.339,-176.715,7.375,148.438
C05103=1195.136,292.980,-68.309,-176.717,7.373,148.438
C05104=1195.140,292.732,-68.280,-176.720,7.370,148.438
C05105=1195.144,292.483,-68.251,-176.723,7.367,148.438
C05106=1195.149,292.235,-68.221,-176.725,7.365,148.438
C05107=1195.153,291.987,-68.192,-176.728,7.362,148.438
C05108=1195.157,291.738,-68.162,-176.731,7.359,148.438
C05109=1195.161,291.490,-68.133,-176.733,7.357,148.438
C05110=1195.166,291.243,-68.104,-176.736,7.354,148.438
C05111=1195.170,290.994,-68.075,-176.738,7.351,148.438
C05112=1195.175,290.745,-68.045,-176.740,7.349,148.438
C05113=1195.179,290.497,-68.016,-176.743,7.346,148.438
C05114=1195.183,290.249,-67.987,-176.746,7.343,148.438
C05115=1195.187,290.001,-67.957,-176.748,7.340,148.438
C05116=1195.192,289.752,-67.929,-176.751,7.337,148.438
C05117=1195.196,289.504,-67.899,-176.753,7.335,148.439
C05118=1195.201,289.256,-67.870,-176.755,7.332,148.439
C05119=1195.205,288.982,-67.838,-176.758,7.329,148.439
C05120=1195.209,288.707,-67.805,-176.761,7.327,148.439
C05121=1195.215,288.432,-67.773,-176.764,7.324,148.439
C05122=1195.220,288.158,-67.742,-176.767,7.321,148.439
C05123=1195.224,287.910,-67.712,-176.769,7.318,148.439
C05124=1195.228,287.662,-67.683,-176.772,7.315,148.439
C05125=1195.232,287.413,-67.654,-176.774,7.312,148.439
C05126=1195.237,287.165,-67.625,-176.777,7.309,148.439
C05127=1195.241,286.917,-67.596,-176.779,7.307,148.439
C05128=1195.245,286.668,-67.567,-176.782,7.304,148.439
C05129=1195.249,286.420,-67.538,-176.785,7.301,148.439
C05130=1195.254,286.172,-67.509,-176.787,7.299,148.439
C05131=1195.259,285.924,-67.480,-176.790,7.296,148.439
C05132=1195.262,285.676,-67.451,-176.792,7.294,148.440
C05133=1195.267,285.427,-67.422,-176.795,7.291,148.440
C05134=1195.271,285.179,-67.393,-176.797,7.288,148.440
C05135=1195.276,284.930,-67.365,-176.800,7.286,148.440
C05136=1195.280,284.682,-67.335,-176.802,7.283,148.440
C05137=1195.284,284.434,-67.307,-176.805,7.280,148.440
C05138=1195.289,284.186,-67.278,-176.808,7.278,148.440
C05139=1195.293,283.937,-67.249,-176.810,7.275,148.440
C05140=1195.298,283.689,-67.220,-176.813,7.273,148.440
C05141=1195.302,283.441,-67.192,-176.815,7.270,148.440
C05142=1195.306,283.193,-67.162,-176.818,7.267,148.440
C05143=1195.310,282.944,-67.134,-176.820,7.265,148.440
C05144=1195.315,282.696,-67.105,-176.823,7.262,148.440
C05145=1195.319,282.448,-67.076,-176.825,7.259,148.440
C05146=1195.323,282.199,-67.048,-176.828,7.257,148.441
C05147=1195.328,281.951,-67.019,-176.831,7.254,148.441
C05148=1195.332,281.702,-66.991,-176.833,7.252,148.441
C05149=1195.337,281.455,-66.961,-176.836,7.249,148.441
C05150=1195.341,281.206,-66.933,-176.838,7.246,148.441
C05151=1195.345,280.957,-66.905,-176.841,7.243,148.441
C05152=1195.350,280.710,-66.875,-176.844,7.241,148.441
C05153=1195.354,280.461,-66.847,-176.846,7.239,148.441
C05154=1195.358,280.212,-66.819,-176.849,7.236,148.441
C05155=1195.363,279.965,-66.789,-176.851,7.233,148.441
C05156=1195.366,279.716,-66.761,-176.853,7.230,148.441
C05157=1195.371,279.467,-66.733,-176.856,7.228,148.441
C05158=1195.376,279.219,-66.704,-176.859,7.225,148.442
C05159=1195.379,278.971,-66.675,-176.861,7.222,148.442
C05160=1195.384,278.723,-66.647,-176.864,7.220,148.442
C05161=1195.388,278.474,-66.619,-176.866,7.217,148.442
C05162=1195.393,278.226,-66.590,-176.868,7.215,148.442
C05163=1195.397,277.978,-66.562,-176.871,7.212,148.442
C05164=1195.401,277.729,-66.533,-176.874,7.210,148.442
C05165=1195.406,277.482,-66.505,-176.876,7.207,148.442
C05166=1195.410,277.233,-66.476,-176.879,7.204,148.442
C05167=1195.414,276.984,-66.448,-176.881,7.202,148.442
C05168=1195.419,276.736,-66.420,-176.884,7.199,148.442
C05169=1195.423,276.487,-66.392,-176.887,7.197,148.443
C05170=1195.428,276.239,-66.363,-176.889,7.194,148.443
C05171=1195.431,275.991,-66.334,-176.892,7.192,148.443
C05172=1195.436,275.743,-66.306,-176.894,7.189,148.443
C05173=1195.440,275.494,-66.278,-176.897,7.186,148.443
C05174=1195.445,275.246,-66.250,-176.900,7.184,148.443
C05175=1195.449,274.998,-66.221,-176.902,7.181,148.443
C05176=1195.454,274.750,-66.193,-176.904,7.179,148.443
C05177=1195.458,274.501,-66.165,-176.907,7.176,148.443
C05178=1195.463,274.253,-66.137,-176.910,7.174,148.444
C05179=1195.467,274.004,-66.108,-176.912,7.171,148.444
C05180=1195.471,273.756,-66.081,-176.915,7.169,148.444
C05181=1195.475,273.507,-66.052,-176.917,7.166,148.444
C05182=1195.480,273.260,-66.024,-176.919,7.164,148.444
C05183=1195.484,273.011,-65.995,-176.923,7.161,148.444
C05184=1195.489,272.763,-65.968,-176.925,7.158,148.444
C05185=1195.492,272.514,-65.939,-176.928,7.156,148.444
C05186=1195.498,272.265,-65.912,-176.930,7.153,148.444
C05187=1195.501,272.017,-65.884,-176.933,7.151,148.445
C05188=1195.507,271.769,-65.855,-176.936,7.148,148.445
C05189=1195.510,271.520,-65.827,-176.938,7.146,148.445
C05190=1195.515,271.272,-65.799,-176.940,7.143,148.445
C05191=1195.519,271.023,-65.771,-176.943,7.141,148.445
C05192=1195.524,270.775,-65.743,-176.946,7.138,148.445
C05193=1195.528,270.526,-65.715,-176.948,7.136,148.445
C05194=1195.532,270.278,-65.688,-176.951,7.133,148.445
C05195=1195.537,270.030,-65.659,-176.953,7.131,148.445
C05196=1195.541,269.782,-65.631,-176.956,7.128,148.446
C05197=1195.545,269.534,-65.603,-176.958,7.126,148.446
C05198=1195.550,269.284,-65.575,-176.961,7.123,148.446
C05199=1195.554,269.036,-65.548,-176.963,7.121,148.446
C05200=1195.559,268.788,-65.520,-176.966,7.118,148.446
C05201=1195.562,268.540,-65.492,-176.968,7.116,148.446
C05202=1195.568,268.291,-65.464,-176.971,7.113,148.446
C05203=1195.572,268.042,-65.436,-176.974,7.111,148.446
C05204=1195.576,267.795,-65.408,-176.976,7.108,148.446
C05205=1195.581,267.546,-65.381,-176.979,7.106,148.447
C05206=1195.585,267.297,-65.352,-176.982,7.103,148.447
C05207=1195.589,267.049,-65.325,-176.984,7.101,148.447
C05208=1195.594,266.801,-65.297,-176.987,7.098,148.447
C05209=1195.598,266.552,-65.269,-176.989,7.096,148.447
C05210=1195.602,266.304,-65.242,-176.992,7.093,148.447
C05211=1195.607,266.055,-65.214,-176.994,7.091,148.447
C05212=1195.611,265.807,-65.186,-176.997,7.088,148.448
C05213=1195.616,265.559,-65.159,-176.999,7.086,148.448
C05214=1195.620,265.310,-65.131,-177.002,7.083,148.448
C05215=1195.624,265.061,-65.103,-177.005,7.081,148.448
C05216=1195.629,264.814,-65.076,-177.007,7.078,148.448
C05217=1195.632,264.565,-65.048,-177.010,7.076,148.448
C05218=1195.638,264.316,-65.020,-177.012,7.073,148.448
C05219=1195.642,264.068,-64.992,-177.015,7.071,148.448
C05220=1195.647,263.820,-64.965,-177.018,7.068,148.449
C05221=1195.651,263.571,-64.937,-177.020,7.066,148.449
C05222=1195.655,263.323,-64.910,-177.023,7.063,148.449
C05223=1195.660,263.050,-64.880,-177.025,7.061,148.449
C05224=1195.664,262.777,-64.849,-177.028,7.058,148.449
C05225=1195.670,262.504,-64.819,-177.031,7.055,148.449
C05226=1195.674,262.231,-64.788,-177.034,7.053,148.450
C05227=1195.679,261.983,-64.761,-177.036,7.051,148.450
C05228=1195.683,261.735,-64.734,-177.039,7.048,148.450
C05229=1195.688,261.486,-64.707,-177.042,7.046,148.450
C05230=1195.692,261.237,-64.679,-177.044,7.043,148.450
C05231=1195.696,260.989,-64.651,-177.047,7.041,148.450
C05232=1195.701,260.741,-64.624,-177.050,7.038,148.450
C05233=1195.706,260.492,-64.597,-177.052,7.036,148.450
C05234=1195.709,260.244,-64.569,-177.055,7.033,148.451
C05235=1195.714,259.995,-64.542,-177.057,7.031,148.451
C05236=1195.719,259.747,-64.515,-177.059,7.029,148.451
C05237=1195.723,259.499,-64.487,-177.063,7.026,148.451
C05238=1195.727,259.250,-64.460,-177.065,7.024,148.451
C05239=1195.731,259.001,-64.433,-177.067,7.021,148.451
C05240=1195.736,258.753,-64.406,-177.070,7.019,148.452
C05241=1195.740,258.505,-64.378,-177.073,7.016,148.452
C05242=1195.745,258.257,-64.351,-177.075,7.014,148.452
C05243=1195.749,258.007,-64.324,-177.078,7.011,148.452
C05244=1195.753,257.759,-64.297,-177.080,7.009,148.452
C05245=1195.758,257.510,-64.270,-177.083,7.007,148.452
C05246=1195.762,257.262,-64.242,-177.086,7.004,148.452
C05247=1195.767,257.014,-64.215,-177.088,7.002,148.453
C05248=1195.772,256.765,-64.188,-177.091,6.999,148.453
C05249=1195.775,256.517,-64.161,-177.093,6.997,148.453
C05250=1195.780,256.268,-64.134,-177.096,6.994,148.453
C05251=1195.784,256.020,-64.107,-177.099,6.992,148.453
C05252=1195.789,255.771,-64.080,-177.101,6.990,148.453
C05253=1195.794,255.523,-64.053,-177.104,6.988,148.454
C05254=1195.798,255.274,-64.026,-177.106,6.985,148.454
C05255=1195.803,255.026,-63.998,-177.109,6.983,148.454
C05256=1195.806,254.777,-63.971,-177.111,6.981,148.454
C05257=1195.811,254.529,-63.944,-177.114,6.978,148.454
C05258=1195.815,254.280,-63.917,-177.117,6.976,148.454
C05259=1195.820,254.032,-63.890,-177.119,6.974,148.455
C05260=1195.824,253.784,-63.864,-177.122,6.971,148.455
C05261=1195.829,253.535,-63.836,-177.124,6.969,148.455
C05262=1195.833,253.287,-63.809,-177.126,6.967,148.455
C05263=1195.838,253.038,-63.782,-177.130,6.964,148.455
C05264=1195.841,252.789,-63.756,-177.132,6.962,148.455
C05265=1195.846,252.541,-63.728,-177.135,6.959,148.456
C05266=1195.851,252.292,-63.702,-177.137,6.957,148.456
C05267=1195.856,252.043,-63.675,-177.140,6.955,148.456
C05268=1195.859,251.795,-63.649,-177.142,6.952,148.456
C05269=1195.864,251.547,-63.622,-177.145,6.950,148.456
C05270=1195.869,251.298,-63.594,-177.148,6.947,148.456
C05271=1195.873,251.050,-63.568,-177.150,6.945,148.457
C05272=1195.877,250.801,-63.541,-177.153,6.943,148.457
C05273=1195.882,250.553,-63.514,-177.155,6.940,148.457
C05274=1195.887,250.304,-63.487,-177.158,6.938,148.457
C05275=1195.891,250.056,-63.461,-177.160,6.936,148.457
C05276=1195.896,249.807,-63.434,-177.163,6.933,148.458
C05277=1195.899,249.559,-63.408,-177.165,6.931,148.458
C05278=1195.904,249.310,-63.380,-177.169,6.929,148.458
C05279=1195.909,249.062,-63.353,-177.171,6.926,148.458
C05280=1195.913,248.813,-63.328,-177.173,6.924,148.458
C05281=1195.918,248.565,-63.301,-177.176,6.922,148.458
C05282=1195.922,248.316,-63.274,-177.178,6.919,148.459
C05283=1195.926,248.068,-63.247,-177.181,6.918,148.459
C05284=1195.931,247.819,-63.221,-177.184,6.915,148.459
C05285=1195.935,247.571,-63.194,-177.186,6.913,148.459
C05286=1195.940,247.322,-63.167,-177.189,6.910,148.459
C05287=1195.945,247.073,-63.141,-177.192,6.908,148.460
C05288=1195.949,246.825,-63.114,-177.194,6.906,148.460
C05289=1195.953,246.576,-63.087,-177.197,6.903,148.460
C05290=1195.958,246.328,-63.062,-177.199,6.901,148.460
C05291=1195.962,246.079,-63.035,-177.202,6.899,148.460
C05292=1195.966,245.831,-63.008,-177.204,6.896,148.460
C05293=1195.971,245.582,-62.982,-177.207,6.894,148.461
C05294=1195.975,245.334,-62.955,-177.209,6.892,148.461
C05295=1195.980,245.084,-62.929,-177.212,6.889,148.461
C05296=1195.984,244.836,-62.902,-177.215,6.887,148.461
C05297=1195.989,244.588,-62.875,-177.217,6.885,148.462
C05298=1195.993,244.339,-62.850,-177.220,6.882,148.462
C05299=1195.997,244.090,-62.823,-177.223,6.881,148.462
C05300=1196.002,243.842,-62.797,-177.225,6.878,148.462
C05301=1196.006,243.593,-62.770,-177.228,6.876,148.462
C05302=1196.011,243.344,-62.744,-177.230,6.874,148.462
C05303=1196.015,243.097,-62.718,-177.233,6.872,148.463
C05304=1196.020,242.848,-62.692,-177.235,6.869,148.463
C05305=1196.024,242.600,-62.665,-177.238,6.867,148.463
C05306=1196.029,242.350,-62.639,-177.240,6.865,148.463
C05307=1196.033,242.102,-62.612,-177.243,6.862,148.463
C05308=1196.038,241.853,-62.586,-177.246,6.860,148.464
C05309=1196.042,241.604,-62.560,-177.248,6.858,148.464
C05310=1196.046,241.356,-62.534,-177.251,6.855,148.464
C05311=1196.051,241.107,-62.507,-177.254,6.853,148.464
C05312=1196.055,240.860,-62.481,-177.256,6.851,148.465
C05313=1196.060,240.611,-62.456,-177.259,6.848,148.465
C05314=1196.065,240.362,-62.429,-177.262,6.847,148.465
C05315=1196.068,240.113,-62.403,-177.264,6.845,148.465
C05316=1196.073,239.864,-62.376,-177.266,6.843,148.465
C05317=1196.078,239.615,-62.351,-177.269,6.840,148.465
C05318=1196.082,239.368,-62.325,-177.272,6.838,148.466
C05319=1196.087,239.119,-62.298,-177.274,6.836,148.466
C05320=1196.091,238.870,-62.272,-177.277,6.833,148.466
C05321=1196.095,238.622,-62.246,-177.280,6.831,148.466
C05322=1196.100,238.373,-62.220,-177.282,6.829,148.467
C05323=1196.104,238.124,-62.194,-177.285,6.826,148.467
C05324=1196.109,237.876,-62.168,-177.287,6.824,148.467
C05325=1196.113,237.628,-62.142,-177.290,6.822,148.467
C05326=1196.118,237.379,-62.116,-177.292,6.820,148.467
C05327=1196.123,237.107,-62.088,-177.295,6.818,148.468
C05328=1196.128,236.836,-62.059,-177.298,6.815,148.468
C05329=1196.133,236.564,-62.031,-177.301,6.813,148.468
C05330=1196.137,236.292,-62.003,-177.304,6.810,148.468
C05331=1196.141,236.044,-61.977,-177.306,6.808,148.469
C05332=1196.147,235.796,-61.951,-177.309,6.806,148.469
C05333=1196.151,235.547,-61.925,-177.312,6.803,148.469
C05334=1196.155,235.298,-61.899,-177.314,6.802,148.469
C05335=1196.159,235.049,-61.873,-177.317,6.799,148.469
C05336=1196.164,234.801,-61.848,-177.319,6.798,148.470
C05337=1196.169,234.552,-61.822,-177.322,6.795,148.470
C05338=1196.173,234.303,-61.796,-177.325,6.793,148.470
C05339=1196.178,234.054,-61.770,-177.327,6.791,148.470
C05340=1196.182,233.807,-61.744,-177.330,6.788,148.471
C05341=1196.186,233.558,-61.718,-177.333,6.786,148.471
C05342=1196.191,233.309,-61.693,-177.335,6.784,148.471
C05343=1196.196,233.061,-61.667,-177.337,6.782,148.471
C05344=1196.200,232.812,-61.641,-177.341,6.779,148.472
C05345=1196.205,232.563,-61.615,-177.343,6.777,148.472
C05346=1196.209,232.315,-61.589,-177.345,6.775,148.472
C05347=1196.214,232.066,-61.564,-177.348,6.774,148.472
C05348=1196.218,231.818,-61.538,-177.351,6.771,148.472
C05349=1196.222,231.569,-61.512,-177.353,6.769,148.473
C05350=1196.227,231.320,-61.488,-177.356,6.767,148.473
C05351=1196.231,231.071,-61.462,-177.358,6.765,148.473
C05352=1196.236,230.823,-61.436,-177.361,6.762,148.473
C05353=1196.241,230.574,-61.411,-177.364,6.760,148.474
C05354=1196.245,230.326,-61.385,-177.366,6.758,148.474
C05355=1196.249,230.077,-61.359,-177.369,6.756,148.474
C05356=1196.255,229.828,-61.333,-177.372,6.753,148.474
C05357=1196.259,229.580,-61.308,-177.374,6.752,148.475
C05358=1196.263,229.331,-61.282,-177.377,6.750,148.475
C05359=1196.268,229.082,-61.257,-177.379,6.748,148.475
C05360=1196.272,228.833,-61.232,-177.382,6.745,148.475
C05361=1196.277,228.584,-61.206,-177.385,6.743,148.476
C05362=1196.281,228.336,-61.180,-177.387,6.741,148.476
C05363=1196.285,228.088,-61.155,-177.390,6.739,148.476
C05364=1196.290,227.839,-61.131,-177.392,6.737,148.476
C05365=1196.294,227.590,-61.105,-177.395,6.734,148.476
C05366=1196.298,227.342,-61.079,-177.398,6.732,148.477
C05367=1196.303,227.093,-61.054,-177.400,6.731,148.477
C05368=1196.308,226.844,-61.029,-177.403,6.728,148.477
C05369=1196.313,226.596,-61.003,-177.406,6.726,148.478
C05370=1196.317,226.347,-60.978,-177.408,6.724,148.478
C05371=1196.321,226.098,-60.952,-177.411,6.722,148.478
C05372=1196.326,225.850,-60.927,-177.413,6.720,148.478
C05373=1196.330,225.601,-60.901,-177.416,6.718,148.479
C05374=1196.335,225.353,-60.876,-177.419,6.715,148.479
C05375=1196.340,225.103,-60.851,-177.421,6.713,148.479
C05376=1196.344,224.855,-60.826,-177.424,6.711,148.479
C05377=1196.348,224.606,-60.801,-177.426,6.709,148.479
C05378=1196.353,224.357,-60.775,-177.429,6.707,148.480
C05379=1196.357,224.109,-60.750,-177.432,6.705,148.480
C05380=1196.362,223.860,-60.725,-177.434,6.703,148.480
C05381=1196.367,223.612,-60.700,-177.437,6.701,148.481
C05382=1196.371,223.362,-60.674,-177.439,6.699,148.481
C05383=1196.375,223.114,-60.650,-177.443,6.696,148.481
C05384=1196.380,222.865,-60.625,-177.445,6.694,148.481
C05385=1196.385,222.617,-60.599,-177.447,6.692,148.482
C05386=1196.389,222.368,-60.574,-177.450,6.691,148.482
C05387=1196.394,222.119,-60.549,-177.452,6.688,148.482
C05388=1196.398,221.871,-60.524,-177.455,6.686,148.482
C05389=1196.403,221.622,-60.499,-177.458,6.684,148.483
C05390=1196.407,221.373,-60.473,-177.461,6.682,148.483
C05391=1196.412,221.125,-60.449,-177.463,6.680,148.483
C05392=1196.416,220.875,-60.424,-177.465,6.678,148.483
C05393=1196.421,220.627,-60.399,-177.469,6.675,148.484
C05394=1196.425,220.378,-60.374,-177.471,6.673,148.484
C05395=1196.430,220.130,-60.348,-177.473,6.671,148.484
C05396=1196.434,219.881,-60.324,-177.476,6.670,148.484
C05397=1196.439,219.633,-60.299,-177.479,6.668,148.485
C05398=1196.443,219.383,-60.274,-177.482,6.665,148.485
C05399=1196.448,219.135,-60.249,-177.484,6.663,148.485
C05400=1196.453,218.887,-60.224,-177.487,6.661,148.486
C05401=1196.457,218.637,-60.199,-177.489,6.659,148.486
C05402=1196.461,218.389,-60.175,-177.492,6.657,148.486
C05403=1196.466,218.140,-60.149,-177.494,6.655,148.486
C05404=1196.471,217.891,-60.125,-177.497,6.653,148.487
C05405=1196.475,217.642,-60.100,-177.500,6.651,148.487
C05406=1196.479,217.394,-60.075,-177.502,6.649,148.487
C05407=1196.485,217.145,-60.050,-177.505,6.647,148.487
C05408=1196.488,216.896,-60.026,-177.508,6.645,148.488
C05409=1196.493,216.647,-60.001,-177.510,6.643,148.488
C05410=1196.498,216.399,-59.975,-177.513,6.640,148.488
C05411=1196.502,216.150,-59.951,-177.516,6.639,148.488
C05412=1196.507,215.902,-59.926,-177.518,6.637,148.489
C05413=1196.511,215.652,-59.902,-177.521,6.635,148.489
C05414=1196.516,215.404,-59.877,-177.524,6.633,148.490
C05415=1196.520,215.155,-59.852,-177.526,6.631,148.490
C05416=1196.525,214.906,-59.827,-177.529,6.628,148.490
C05417=1196.530,214.658,-59.803,-177.532,6.626,148.490
C05418=1196.534,214.409,-59.778,-177.534,6.625,148.491
C05419=1196.539,214.160,-59.754,-177.536,6.622,148.491
C05420=1196.543,213.912,-59.730,-177.539,6.621,148.491
C05421=1196.547,213.663,-59.704,-177.542,6.619,148.491
C05422=1196.552,213.414,-59.680,-177.545,6.616,148.492
C05423=1196.557,213.166,-59.655,-177.548,6.614,148.492
C05424=1196.561,212.916,-59.631,-177.550,6.612,148.492
C05425=1196.566,212.668,-59.606,-177.552,6.610,148.492
C05426=1196.570,212.419,-59.582,-177.555,6.609,148.493
C05427=1196.575,212.170,-59.557,-177.558,6.607,148.493
C05428=1196.579,211.921,-59.533,-177.560,6.605,148.493
C05429=1196.584,211.673,-59.508,-177.563,6.602,148.494
C05430=1196.588,211.424,-59.484,-177.566,6.600,148.494
C05431=1196.593,211.153,-59.457,-177.568,6.598,148.494
C05432=1196.598,210.883,-59.430,-177.572,6.596,148.495
C05433=1196.604,210.613,-59.404,-177.574,6.594,148.495
C05434=1196.608,210.342,-59.377,-177.577,6.592,148.495
C05435=1196.613,210.093,-59.353,-177.580,6.590,148.496
C05436=1196.617,209.845,-59.329,-177.583,6.588,148.496
C05437=1196.622,209.596,-59.304,-177.585,6.585,148.496
C05438=1196.626,209.347,-59.280,-177.588,6.584,148.496
C05439=1196.631,209.098,-59.255,-177.590,6.582,148.497
C05440=1196.636,208.850,-59.231,-177.593,6.580,148.497
C05441=1196.640,208.601,-59.207,-177.596,6.578,148.497
C05442=1196.645,208.352,-59.182,-177.598,6.576,148.498
C05443=1196.649,208.104,-59.158,-177.600,6.574,148.498
C05444=1196.654,207.854,-59.134,-177.604,6.572,148.498
C05445=1196.659,207.606,-59.110,-177.606,6.570,148.498
C05446=1196.663,207.357,-59.086,-177.609,6.568,148.499
C05447=1196.668,207.108,-59.061,-177.611,6.566,148.499
C05448=1196.672,206.860,-59.037,-177.614,6.564,148.499
C05449=1196.677,206.611,-59.013,-177.616,6.562,148.500
C05450=1196.682,206.362,-58.989,-177.619,6.560,148.500
C05451=1196.686,206.113,-58.964,-177.622,6.558,148.500
C05452=1196.690,205.864,-58.940,-177.624,6.557,148.501
C05453=1196.695,205.616,-58.916,-177.627,6.554,148.501
C05454=1196.700,205.367,-58.892,-177.630,6.552,148.501
C05455=1196.704,205.118,-58.868,-177.632,6.550,148.501
C05456=1196.708,204.869,-58.844,-177.635,6.548,148.502
C05457=1196.713,204.620,-58.820,-177.638,6.546,148.502
C05458=1196.718,204.371,-58.796,-177.640,6.545,148.502
C05459=1196.722,204.123,-58.772,-177.643,6.543,148.503
C05460=1196.727,203.874,-58.748,-177.646,6.541,148.503
C05461=1196.732,203.625,-58.724,-177.648,6.539,148.503
C05462=1196.736,203.376,-58.699,-177.650,6.537,148.504
C05463=1196.741,203.127,-58.676,-177.653,6.535,148.504
C05464=1196.745,202.879,-58.652,-177.656,6.533,148.504
C05465=1196.750,202.630,-58.628,-177.659,6.531,148.505
C05466=1196.754,202.381,-58.604,-177.662,6.529,148.505
C05467=1196.759,202.132,-58.580,-177.664,6.527,148.505
C05468=1196.764,201.884,-58.556,-177.667,6.525,148.506
C05469=1196.768,201.634,-58.532,-177.669,6.523,148.506
C05470=1196.772,201.386,-58.508,-177.672,6.521,148.506
C05471=1196.777,201.137,-58.484,-177.674,6.519,148.506
C05472=1196.781,200.888,-58.460,-177.677,6.518,148.507
C05473=1196.786,200.639,-58.437,-177.680,6.516,148.507
